# B&R Automation Studio project TD52 (part 94)

```iecst
	(* W9687 SAFETY - Room ventilation failure - Outlet air louvre group 3 - closed signal not valid *)
	xMsg9687.Enable	   		:= OUT_EG.bSafetyPLC_Active AND bRelModul_ParaSetupOk;			(* SAFETY PLC *)
	xMsg9687.Set	  		:= NOT bAMM_9687;
	xMsg9687.PT	       		:= T#0s;
	xMsg9687.Prio	   		:= 4;
	xMsg9687.RiskClass		:= 4;
	xMsg9687.Reset	   		:= FALSE;
	xMsg9687();
	MM2VIS.bMsg9687			:= xMsg9687.Q;

	(* W9688 SAFETY - Room ventilation failure - Outlet air louvre group 3 - plausibility check failure *)
	xMsg9688.Enable	   		:= OUT_EG.bSafetyPLC_Active AND bRelModul_ParaSetupOk;			(* SAFETY PLC *)
	xMsg9688.Set	  		:= NOT bAMM_9688;
	xMsg9688.PT	       		:= T#0s;
	xMsg9688.Prio	   		:= 4;
	xMsg9688.RiskClass		:= 4;
	xMsg9688.Reset	   		:= FALSE;
	xMsg9688();
	MM2VIS.bMsg9688			:= xMsg9688.Q;

	(* W9689 SAFETY - Room ventilation failure - Outlet air louvre group 4 - closed signal *)
	xMsg9689.Enable	   		:= OUT_EG.bSafetyPLC_Active AND bRelModul_ParaSetupOk;			(* SAFETY PLC *)
	xMsg9689.Set	  		:= NOT bAMM_9689;
	xMsg9689.PT	       		:= T#0s;
	xMsg9689.Prio	   		:= 4;
	xMsg9689.RiskClass		:= 4;
	xMsg9689.Reset	   		:= FALSE;
	xMsg9689();
	MM2VIS.bMsg9689			:= xMsg9689.Q;

	(* W9690 SAFETY - Room ventilation failure - Outlet air louvre group 4 - opened signal not valid *)
	xMsg9690.Enable	   		:= OUT_EG.bSafetyPLC_Active AND bRelModul_ParaSetupOk;			(* SAFETY PLC *)
	xMsg9690.Set	  		:= NOT bAMM_9690;
	xMsg9690.PT	       		:= T#0s;
	xMsg9690.Prio	   		:= 4;
	xMsg9690.RiskClass		:= 4;
	xMsg9690.Reset	   		:= FALSE;
	xMsg9690();
	MM2VIS.bMsg9690			:= xMsg9690.Q;

	(* W9691 SAFETY - Room ventilation failure - Outlet air louvre group 4 - closed signal not valid *)
	xMsg9691.Enable	   		:= OUT_EG.bSafetyPLC_Active AND bRelModul_ParaSetupOk;			(* SAFETY PLC *)
	xMsg9691.Set	  		:= NOT bAMM_9691;
	xMsg9691.PT	       		:= T#0s;
	xMsg9691.Prio	   		:= 4;
	xMsg9691.RiskClass		:= 4;
	xMsg9691.Reset	   		:= FALSE;
	xMsg9691();
	MM2VIS.bMsg9691			:= xMsg9691.Q;

	(* W9692 SAFETY - Room ventilation failure - Outlet air louvre group 4 - plausibility check failure *)
	xMsg9692.Enable	   		:= OUT_EG.bSafetyPLC_Active AND bRelModul_ParaSetupOk;			(* SAFETY PLC *)
	xMsg9692.Set	  		:= NOT bAMM_9692;
	xMsg9692.PT	       		:= T#0s;
	xMsg9692.Prio	   		:= 4;
	xMsg9692.RiskClass		:= 4;
	xMsg9692.Reset	   		:= FALSE;
	xMsg9692();
	MM2VIS.bMsg9692			:= xMsg9692.Q;

	(* W9693 SAFETY - Room ventilation failure - Outlet air louvre group 5 - closed signal *)
	xMsg9693.Enable	   		:= OUT_EG.bSafetyPLC_Active AND bRelModul_ParaSetupOk;			(* SAFETY PLC *)
	xMsg9693.Set	  		:= NOT bAMM_9693;
	xMsg9693.PT	       		:= T#0s;
	xMsg9693.Prio	   		:= 4;
	xMsg9693.RiskClass		:= 4;
	xMsg9693.Reset	   		:= FALSE;
	xMsg9693();
	MM2VIS.bMsg9693			:= xMsg9693.Q;

	(* W9694 SAFETY - Room ventilation failure - Outlet air louvre group 5 - opened signal not valid *)
	xMsg9694.Enable	   		:= OUT_EG.bSafetyPLC_Active AND bRelModul_ParaSetupOk;			(* SAFETY PLC *)
	xMsg9694.Set	  		:= NOT bAMM_9694;
	xMsg9694.PT	       		:= T#0s;
	xMsg9694.Prio	   		:= 4;
	xMsg9694.RiskClass		:= 4;
	xMsg9694.Reset	   		:= FALSE;
	xMsg9694();
	MM2VIS.bMsg9694			:= xMsg9694.Q;

	(* W9695 SAFETY - Room ventilation failure - Outlet air louvre group 5 - closed signal not valid *)
	xMsg9695.Enable	   		:= OUT_EG.bSafetyPLC_Active AND bRelModul_ParaSetupOk;			(* SAFETY PLC *)
	xMsg9695.Set	  		:= NOT bAMM_9695;
	xMsg9695.PT	       		:= T#0s;
	xMsg9695.Prio	   		:= 4;
	xMsg9695.RiskClass		:= 4;
	xMsg9695.Reset	   		:= FALSE;
	xMsg9695();
	MM2VIS.bMsg9695			:= xMsg9695.Q;

	(* W9696 SAFETY - Room ventilation failure - Outlet air louvre group 5 - plausibility check failure *)
	xMsg9696.Enable	   		:= OUT_EG.bSafetyPLC_Active AND bRelModul_ParaSetupOk;			(* SAFETY PLC *)
	xMsg9696.Set	  		:= NOT bAMM_9696;
	xMsg9696.PT	       		:= T#0s;
	xMsg9696.Prio	   		:= 4;
	xMsg9696.RiskClass		:= 4;
	xMsg9696.Reset	   		:= FALSE;
	xMsg9696();
	MM2VIS.bMsg9696			:= xMsg9696.Q;

	(* W9697 SAFETY - Room ventilation failure - Outlet air louvre group 6 - closed signal *)
	xMsg9697.Enable	   		:= OUT_EG.bSafetyPLC_Active AND bRelModul_ParaSetupOk;			(* SAFETY PLC *)
	xMsg9697.Set	  		:= NOT bAMM_9697;
	xMsg9697.PT	       		:= T#0s;
	xMsg9697.Prio	   		:= 4;
	xMsg9697.RiskClass		:= 4;
	xMsg9697.Reset	   		:= FALSE;
	xMsg9697();
	MM2VIS.bMsg9697			:= xMsg9697.Q;

	(* W9698 SAFETY - Room ventilation failure - Outlet air louvre group 6 - opened signal not valid *)
	xMsg9698.Enable	   		:= OUT_EG.bSafetyPLC_Active AND bRelModul_ParaSetupOk;			(* SAFETY PLC *)
	xMsg9698.Set	  		:= NOT bAMM_9698;
	xMsg9698.PT	       		:= T#0s;
	xMsg9698.Prio	   		:= 4;
	xMsg9698.RiskClass		:= 4;
	xMsg9698.Reset	   		:= FALSE;
	xMsg9698();
	MM2VIS.bMsg9698			:= xMsg9698.Q;

	(* W9699 SAFETY - Room ventilation failure - Outlet air louvre group 6 - closed signal not valid *)
	xMsg9699.Enable	   		:= OUT_EG.bSafetyPLC_Active AND bRelModul_ParaSetupOk;			(* SAFETY PLC *)
	xMsg9699.Set	  		:= NOT bAMM_9699;
	xMsg9699.PT	       		:= T#0s;
	xMsg9699.Prio	   		:= 4;
	xMsg9699.RiskClass		:= 4;
	xMsg9699.Reset	   		:= FALSE;
	xMsg9699();
	MM2VIS.bMsg9699			:= xMsg9699.Q;

	(* W9700 SAFETY - Room ventilation failure - Outlet air louvre group 6 - plausibility check failure *)
	xMsg9700.Enable	   		:= OUT_EG.bSafetyPLC_Active AND bRelModul_ParaSetupOk;			(* SAFETY PLC *)
	xMsg9700.Set	  		:= NOT bAMM_9700;
	xMsg9700.PT	       		:= T#0s;
	xMsg9700.Prio	   		:= 4;
	xMsg9700.RiskClass		:= 4;
	xMsg9700.Reset	   		:= FALSE;
	xMsg9700();
	MM2VIS.bMsg9700			:= xMsg9700.Q;

	(* W9701 SAFETY - Release gas valve A for decentral gas addition - output not valid *)
	xMsg9701.Enable	   		:= OUT_EG.bSafetyPLC_Active AND bRelModul_ParaSetupOk;			(* SAFETY PLC *)
	xMsg9701.Set	  		:= NOT bAMM_9701;
	xMsg9701.PT	       		:= T#0s;
	xMsg9701.Prio	   		:= 4;
	xMsg9701.RiskClass		:= 4;
	xMsg9701.Reset	   		:= FALSE;
	xMsg9701();
	MM2VIS.bMsg9701			:= xMsg9701.Q;

	(* W9702 SAFETY - Release gas valve B for decentral gas addition - output not valid *)
	xMsg9702.Enable	   		:= OUT_EG.bSafetyPLC_Active AND bRelModul_ParaSetupOk;			(* SAFETY PLC *)
	xMsg9702.Set	  		:= NOT bAMM_9702;
	xMsg9702.PT	       		:= T#0s;
	xMsg9702.Prio	   		:= 4;
	xMsg9702.RiskClass		:= 4;
	xMsg9702.Reset	   		:= FALSE;
	xMsg9702();
	MM2VIS.bMsg9702			:= xMsg9702.Q;

	(* W9703 SAFETY - Gas safety device for decentral gas addition - signal not valid *)
	xMsg9703.Enable	   		:= OUT_EG.bSafetyPLC_Active AND bRelModul_ParaSetupOk;			(* SAFETY PLC *)
	xMsg9703.Set	  		:= NOT bAMM_9703;
	xMsg9703.PT	       		:= T#0s;
	xMsg9703.Prio	   		:= 4;
	xMsg9703.RiskClass		:= 4;
	xMsg9703.Reset	   		:= FALSE;
	xMsg9703();
	MM2VIS.bMsg9703			:= xMsg9703.Q;

	(* W9704 SAFETY - Gas safety device for decentral gas addition - output not valid *)
	xMsg9704.Enable	   		:= OUT_EG.bSafetyPLC_Active AND bRelModul_ParaSetupOk;			(* SAFETY PLC *)
	xMsg9704.Set	  		:= NOT bAMM_9704;
	xMsg9704.PT	       		:= T#0s;
	xMsg9704.Prio	   		:= 4;
	xMsg9704.RiskClass		:= 4;
	xMsg9704.Reset	   		:= FALSE;
	xMsg9704();
	MM2VIS.bMsg9704			:= xMsg9704.Q;

	(*---------------------------------------------------------------------------*)
	(* operating messages > AMM *)

	(* B2190 Emergency stop push button - module control panel (+A/+MC) *)
	xMsg2190.Enable		:= NOT OUT_EG.bSafetyPLC_Active AND bRelModul_ParaSetupOk;			(* SAFETY PLC *)
	xMsg2190.Set		:= IN_EG.tEmStop_MC.Di;
	xMsg2190.Reset		:= TRUE;
	xMsg2190();
	MM2VIS.bMsg2190		:= xMsg2190.Q;

	(* B2191 Emergency stop push button - module interface panel (+M) *)
	xMsg2191.Enable		:= NOT OUT_EG.bSafetyPLC_Active AND bRelModul_ParaSetupOk;			(* SAFETY PLC *)
	xMsg2191.Set		:= IN_EG.tEmStop_M.Di;
	xMsg2191.Reset		:= TRUE;
	xMsg2191();
	MM2VIS.bMsg2191		:= xMsg2191.Q;

	(* B2192 Emergency stop push button – master control panel (+ST) *)
	xMsg2192.Enable		:= NOT OUT_EG.bSafetyPLC_Active AND bRelModul_ParaSetupOk;			(* SAFETY PLC *)
	xMsg2192.Set		:= IN_EG.tEmStop_ST.Di;
	xMsg2192.Reset		:= TRUE;
	xMsg2192();
	MM2VIS.bMsg2192		:= xMsg2192.Q;

	(* B2193 Emergency stop push button – interlock panel (+IS) *)
	xMsg2193.Enable		:= NOT OUT_EG.bSafetyPLC_Active AND bRelModul_ParaSetupOk;			(* SAFETY PLC *)
	xMsg2193.Set		:= IN_EG.tEmStop_IS.Di;
	xMsg2193.Reset		:= TRUE;
	xMsg2193();
	MM2VIS.bMsg2193		:= xMsg2193.Q;

	(* B2194 Emergency stop push button – thermal reactor control panel (+TS) *)
	xMsg2194.Enable		:= NOT OUT_EG.bSafetyPLC_Active AND bRelModul_ParaSetupOk;			(* SAFETY PLC *)
	xMsg2194.Set		:= IN_EG.tEmStop_TS.Di;
	xMsg2194.Reset		:= TRUE;
	xMsg2194();
	MM2VIS.bMsg2194		:= xMsg2194.Q;

	(* B2195 Emergency stop push button – generator interface panel (+GENI) *)
	xMsg2195.Enable		:= NOT OUT_EG.bSafetyPLC_Active AND bRelModul_ParaSetupOk;			(* SAFETY PLC *)
	xMsg2195.Set		:= IN_EG.tEmStop_GENI.Di;
	xMsg2195.Reset		:= TRUE;
	xMsg2195();
	MM2VIS.bMsg2195		:= xMsg2195.Q;

	(* B2196 Emergency stop push button – engine interface panel bank A (+ENGIA) *)
	xMsg2196.Enable		:= NOT OUT_EG.bSafetyPLC_Active AND bRelModul_ParaSetupOk;			(* SAFETY PLC *)
	xMsg2196.Set		:= IN_EG.tEmStop_ENGIA.Di;
	xMsg2196.Reset		:= TRUE;
	xMsg2196();
	MM2VIS.bMsg2196		:= xMsg2196.Q;

	(* B2197 Emergency stop push button – turbocharger module interface panel (+TCMI) *)
	xMsg2197.Enable		:= NOT OUT_EG.bSafetyPLC_Active AND bRelModul_ParaSetupOk;			(* SAFETY PLC *)
	xMsg2197.Set		:= IN_EG.tEmStop_TCMI.Di;
	xMsg2197.Reset		:= TRUE;
	xMsg2197();
	MM2VIS.bMsg2197		:= xMsg2197.Q;

	(* B2198 Emergency stop push button – jacket water module interface panel (+JWMI) *)
	xMsg2198.Enable		:= NOT OUT_EG.bSafetyPLC_Active AND bRelModul_ParaSetupOk;			(* SAFETY PLC *)
	xMsg2198.Set		:= IN_EG.tEmStop_JWMI.Di;
	xMsg2198.Reset		:= TRUE;
	xMsg2198();
	MM2VIS.bMsg2198		:= xMsg2198.Q;

	(* B2199 Emergency stop push button – oil module interface panel (+OILMI) *)
	xMsg2199.Enable		:= NOT OUT_EG.bSafetyPLC_Active AND bRelModul_ParaSetupOk;			(* SAFETY PLC *)
	xMsg2199.Set		:= IN_EG.tEmStop_OILMI.Di;
	xMsg2199.Reset		:= TRUE;
	xMsg2199();
	MM2VIS.bMsg2199		:= xMsg2199.Q;

	(* B2200 Emergency stop push button – exhaust gas after treatment control panel (+SCR) *)
	xMsg2200.Enable		:= NOT OUT_EG.bSafetyPLC_Active AND bRelModul_ParaSetupOk;			(* SAFETY PLC *)
	xMsg2200.Set		:= IN_EG.tEmStop_SCR.Di;
	xMsg2200.Reset		:= TRUE;
	xMsg2200();
	MM2VIS.bMsg2200		:= xMsg2200.Q;

	(* B2804 measuring signal failure main bearing temperature xx *)
	xMsg2804.Enable		:= TRUE;
	xMsg2804.Set		:= bOpM_T_MBearing_Ms;
	xMsg2804.Reset		:= TRUE;
	xMsg2804();
	MM2VIS.bMsg2804		:= xMsg2804.Q;

	(* B2805 main bearing temperature high *)
	xMsg2805.Enable		:= TRUE;
	xMsg2805.Set		:= bOpM_T_MBearing_Hi;
	xMsg2805.Reset		:= TRUE;
	xMsg2805();
	MM2VIS.bMsg2805		:= xMsg2805.Q;

	(* B2806 measuring signal failure conrod bearing temperature xx *)
	xMsg2806.Enable		:= TRUE;
	xMsg2806.Set		:= bOpM_T_CBearing_Ms;
	xMsg2806.Reset		:= TRUE;
	xMsg2806();
	MM2VIS.bMsg2806		:= xMsg2806.Q;

	(* B2807 conrod bearing temperature high *)
	xMsg2807.Enable		:= TRUE;
	xMsg2807.Set		:= bOpM_T_CBearing_Hi;
	xMsg2807.Reset		:= TRUE;
	xMsg2807();
	MM2VIS.bMsg2807		:= xMsg2807.Q;

	(* B2822 conrod bearing signal intensity minimum *)
	xMsg2822.Enable		:= TRUE;
	xMsg2822.Set		:= bOpM_T_CBearing_Sig_Lo;
	xMsg2822.Reset		:= TRUE;
	xMsg2822();
	MM2VIS.bMsg2822		:= xMsg2822.Q;

	(* B2904 main bearing temperature - positive MEDIAN deviation maximum *)
	xMsg2904.Enable		:= TRUE;
	xMsg2904.Set		:= bOpM_T_MBearing_MDev_HiHi;
	xMsg2904.Reset		:= TRUE;
	xMsg2904();
	MM2VIS.bMsg2904		:= xMsg2904.Q;

	(* B2905 conrod bearing temperature - positive MEDIAN deviation maximum *)
	xMsg2905.Enable		:= TRUE;
	xMsg2905.Set		:= bOpM_T_CBearing_MDev_HiHi;
	xMsg2905.Reset		:= TRUE;
	xMsg2905();
	MM2VIS.bMsg2905		:= xMsg2905.Q;

	(* B2909 Conrod bearing temperature calibration successful *)
	xTOF_Calib_Ok(IN 	:= bOpM_T_CBearing_Calib_Ok, PT := T#1s);		(* increase message time from 100ms to 1 s for HMI *)

	xMsg2909.Enable		:= TRUE;
	xMsg2909.Set		:= xTOF_Calib_Ok.Q;
	xMsg2909.Reset		:= TRUE;
	xMsg2909();
	MM2VIS.bMsg2909		:= xMsg2909.Q;

	(* B2958 main bearing temperature - negative MEDIAN deviation maximum *)
	xMsg2958.Enable		:= TRUE;
	xMsg2958.Set		:= bOpM_T_MBearing_MDev_Lo;
	xMsg2958.Reset		:= TRUE;
	xMsg2958();
	MM2VIS.bMsg2958		:= xMsg2958.Q;

	(* B2959 conrod bearing temperature - negative MEDIAN deviation maximum *)
	xMsg2959.Enable		:= TRUE;
	xMsg2959.Set		:= bOpM_T_CBearing_MDev_Lo;
	xMsg2959.Reset		:= TRUE;
	xMsg2959();
	MM2VIS.bMsg2959		:= xMsg2959.Q;

	(* B2981 PU scuffing detection *)
	xMsg2981.Enable		:= Para.bPUscf_Ena;
	xMsg2981.Set		:= bOpM_PUscuff AND bAMM_PUscuff;
	xMsg2981.Reset		:= TRUE;
	xMsg2981();
	MM2VIS.bMsg2981		:= xMsg2981.Q;

	(* B9038 Emergency stop push button – exhaust gas scavenging system control panel (+TCMSCAV) *)
	xMsg9038.Enable		:= NOT OUT_EG.bSafetyPLC_Active AND bRelModul_ParaSetupOk;			(* SAFETY PLC *)
	xMsg9038.Set		:= IN_EG.tEmStop_TCMSCAV.Di;
	xMsg9038.Reset		:= TRUE;
	xMsg9038();
	MM2VIS.bMsg9038		:= xMsg9038.Q;

	(*---------------------------------------------------------------------------*)
	(* general alarms for further module operations *)
	bGnlTrip1 	:= OUT_EG.tEG2AB.bGnlTrip1 		OR IN_EG.tAB2EG.bGnlTrip1;
	bGnlTrip2 	:= OUT_EG.tEG2AB.bGnlTrip2 		OR IN_EG.tAB2EG.bGnlTrip2;
	bGnlTrip3 	:= OUT_EG.tEG2AB.bGnlTrip3 		OR IN_EG.tAB2EG.bGnlTrip3;
	bGnlWarning := OUT_EG.tEG2AB.bGnlWarning	OR IN_EG.tAB2EG.bGnlWarning;
	bGnlTrip	:= bGnlTrip1 OR bGnlTrip2 OR bGnlTrip3;
	(*****************************************************************************)
END_PROGRAM
```

#### MsgEGInit.st - Cyclic code
```iecst
(*******************************************************************************
Msg_EG	 			 alarms generation MM_EngineGeneral

This code is confidential and proprietary to the INNIO Company.
It may not be used in any form, or reproduced in any manner,
without written permission of the INNIO Company.
Copyright, INNIO Company, 2019

Instructions FOR use:
--------------------
1) declare alarm with function block "Msg"

2) use template to create a new alarm, substitue 0000 by message number:

	xMsg0000.Num		:=	0000;					alarm number
	xMsg0000.AmmSysAdr	:=  iAdrAmmBase2MM;			do not change
	xMsg0000.AmmOutAdr	:=  iAdrMM2AmmBase;			do not change

3) 	set alarm number

(*******************************************************************************)
PROGRAM _INIT

	iAdrAmmBase2MM		:= ADR(IN_EG.tAB2EG);
	iAdrMM2AmmBase		:= ADR(OUT_EG.tEG2AB);

	(*---------------------------------------------------------------------------*)

	xMsg1026.Num		:= 1026;
	xMsg1026.AmmInAdr	:= iAdrAmmBase2MM;
	xMsg1026.AmmOutAdr	:= iAdrMM2AmmBase;

	xMsg1031.Num		:= 1031;
	xMsg1031.AmmInAdr	:= iAdrAmmBase2MM;
	xMsg1031.AmmOutAdr	:= iAdrMM2AmmBase;

	xMsg1056.Num		:= 1056;
	xMsg1056.AmmInAdr	:= iAdrAmmBase2MM;
	xMsg1056.AmmOutAdr	:= iAdrMM2AmmBase;

	xMsg1168.Num		:= 1168;
	xMsg1168.AmmInAdr	:= iAdrAmmBase2MM;
	xMsg1168.AmmOutAdr	:= iAdrMM2AmmBase;

	xMsg2190.Num		:= 2190;
	xMsg2190.AmmInAdr	:= iAdrAmmBase2MM;
	xMsg2190.AmmOutAdr	:= iAdrMM2AmmBase;

	xMsg2191.Num		:= 2191;
	xMsg2191.AmmInAdr	:= iAdrAmmBase2MM;
	xMsg2191.AmmOutAdr	:= iAdrMM2AmmBase;

	xMsg2192.Num		:= 2192;
	xMsg2192.AmmInAdr	:= iAdrAmmBase2MM;
	xMsg2192.AmmOutAdr	:= iAdrMM2AmmBase;

	xMsg2193.Num		:= 2193;
	xMsg2193.AmmInAdr	:= iAdrAmmBase2MM;
	xMsg2193.AmmOutAdr	:= iAdrMM2AmmBase;

	xMsg2194.Num		:= 2194;
	xMsg2194.AmmInAdr	:= iAdrAmmBase2MM;
	xMsg2194.AmmOutAdr	:= iAdrMM2AmmBase;

	xMsg2195.Num		:= 2195;
	xMsg2195.AmmInAdr	:= iAdrAmmBase2MM;
	xMsg2195.AmmOutAdr	:= iAdrMM2AmmBase;

	xMsg2196.Num		:= 2196;
	xMsg2196.AmmInAdr	:= iAdrAmmBase2MM;
	xMsg2196.AmmOutAdr	:= iAdrMM2AmmBase;

	xMsg2197.Num		:= 2197;
	xMsg2197.AmmInAdr	:= iAdrAmmBase2MM;
	xMsg2197.AmmOutAdr	:= iAdrMM2AmmBase;

	xMsg2198.Num		:= 2198;
	xMsg2198.AmmInAdr	:= iAdrAmmBase2MM;
	xMsg2198.AmmOutAdr	:= iAdrMM2AmmBase;

	xMsg2199.Num		:= 2199;
	xMsg2199.AmmInAdr	:= iAdrAmmBase2MM;
	xMsg2199.AmmOutAdr	:= iAdrMM2AmmBase;

	xMsg2200.Num		:= 2200;
	xMsg2200.AmmInAdr	:= iAdrAmmBase2MM;
	xMsg2200.AmmOutAdr	:= iAdrMM2AmmBase;

	xMsg2227.Num		:= 2227;
	xMsg2227.AmmInAdr	:= iAdrAmmBase2MM;
	xMsg2227.AmmOutAdr	:= iAdrMM2AmmBase;

	xMsg2228.Num		:= 2228;
	xMsg2228.AmmInAdr	:= iAdrAmmBase2MM;
	xMsg2228.AmmOutAdr	:= iAdrMM2AmmBase;

	xMsg2229.Num		:= 2229;
	xMsg2229.AmmInAdr	:= iAdrAmmBase2MM;
	xMsg2229.AmmOutAdr	:= iAdrMM2AmmBase;

	xMsg2230.Num		:= 2230;
	xMsg2230.AmmInAdr	:= iAdrAmmBase2MM;
	xMsg2230.AmmOutAdr	:= iAdrMM2AmmBase;

	xMsg2232.Num		:= 2232;
	xMsg2232.AmmInAdr	:= iAdrAmmBase2MM;
	xMsg2232.AmmOutAdr	:= iAdrMM2AmmBase;

	xMsg2270.Num		:= 2270;
	xMsg2270.AmmInAdr	:= iAdrAmmBase2MM;
	xMsg2270.AmmOutAdr	:= iAdrMM2AmmBase;

	xMsg2285.Num		:= 2285;
	xMsg2285.AmmInAdr	:= iAdrAmmBase2MM;
	xMsg2285.AmmOutAdr	:= iAdrMM2AmmBase;

	xMsg2286.Num		:= 2286;
	xMsg2286.AmmInAdr	:= iAdrAmmBase2MM;
	xMsg2286.AmmOutAdr	:= iAdrMM2AmmBase;

	xMsg2300.Num		:= 2300;
	xMsg2300.AmmInAdr	:= iAdrAmmBase2MM;
	xMsg2300.AmmOutAdr	:= iAdrMM2AmmBase;

	xMsg2362.Num		:= 2362;
	xMsg2362.AmmInAdr	:= iAdrAmmBase2MM;
	xMsg2362.AmmOutAdr	:= iAdrMM2AmmBase;

	xMsg2383.Num		:= 2383;
	xMsg2383.AmmInAdr	:= iAdrAmmBase2MM;
	xMsg2383.AmmOutAdr	:= iAdrMM2AmmBase;

	xMsg2384.Num		:= 2384;
	xMsg2384.AmmInAdr	:= iAdrAmmBase2MM;
	xMsg2384.AmmOutAdr	:= iAdrMM2AmmBase;

	xMsg2385.Num		:= 2385;
	xMsg2385.AmmInAdr	:= iAdrAmmBase2MM;
	xMsg2385.AmmOutAdr	:= iAdrMM2AmmBase;

	xMsg2386.Num		:= 2386;
	xMsg2386.AmmInAdr	:= iAdrAmmBase2MM;
	xMsg2386.AmmOutAdr	:= iAdrMM2AmmBase;

	xMsg2387.Num		:= 2387;
	xMsg2387.AmmInAdr	:= iAdrAmmBase2MM;
	xMsg2387.AmmOutAdr	:= iAdrMM2AmmBase;

	xMsg2388.Num		:= 2388;
	xMsg2388.AmmInAdr	:= iAdrAmmBase2MM;
	xMsg2388.AmmOutAdr	:= iAdrMM2AmmBase;

	xMsg2389.Num		:= 2389;
	xMsg2389.AmmInAdr	:= iAdrAmmBase2MM;
	xMsg2389.AmmOutAdr	:= iAdrMM2AmmBase;

	xMsg2390.Num		:= 2390;
	xMsg2390.AmmInAdr	:= iAdrAmmBase2MM;
	xMsg2390.AmmOutAdr	:= iAdrMM2AmmBase;

	xMsg2391.Num		:= 2391;
	xMsg2391.AmmInAdr	:= iAdrAmmBase2MM;
	xMsg2391.AmmOutAdr	:= iAdrMM2AmmBase;

	xMsg2392.Num		:= 2392;
	xMsg2392.AmmInAdr	:= iAdrAmmBase2MM;
	xMsg2392.AmmOutAdr	:= iAdrMM2AmmBase;

	xMsg2393.Num		:= 2393;
	xMsg2393.AmmInAdr	:= iAdrAmmBase2MM;
	xMsg2393.AmmOutAdr	:= iAdrMM2AmmBase;

	xMsg2394.Num		:= 2394;
	xMsg2394.AmmInAdr	:= iAdrAmmBase2MM;
	xMsg2394.AmmOutAdr	:= iAdrMM2AmmBase;

	xMsg2395.Num		:= 2395;
	xMsg2395.AmmInAdr	:= iAdrAmmBase2MM;
	xMsg2395.AmmOutAdr	:= iAdrMM2AmmBase;

	xMsg2396.Num		:= 2396;
	xMsg2396.AmmInAdr	:= iAdrAmmBase2MM;
	xMsg2396.AmmOutAdr	:= iAdrMM2AmmBase;

	xMsg2397.Num		:= 2397;
	xMsg2397.AmmInAdr	:= iAdrAmmBase2MM;
	xMsg2397.AmmOutAdr	:= iAdrMM2AmmBase;

	xMsg2398.Num		:= 2398;
	xMsg2398.AmmInAdr	:= iAdrAmmBase2MM;
	xMsg2398.AmmOutAdr	:= iAdrMM2AmmBase;

	xMsg2542.Num		:= 2542;
	xMsg2542.AmmInAdr	:= iAdrAmmBase2MM;
	xMsg2542.AmmOutAdr	:= iAdrMM2AmmBase;

	xMsg2544.Num		:= 2544;
	xMsg2544.AmmInAdr	:= iAdrAmmBase2MM;
	xMsg2544.AmmOutAdr	:= iAdrMM2AmmBase;

	xMsg2552.Num		:= 2552;
	xMsg2552.AmmInAdr	:= iAdrAmmBase2MM;
	xMsg2552.AmmOutAdr	:= iAdrMM2AmmBase;

	xMsg2553.Num		:= 2553;
	xMsg2553.AmmInAdr	:= iAdrAmmBase2MM;
	xMsg2553.AmmOutAdr	:= iAdrMM2AmmBase;

	xMsg2561.Num		:= 2561;
	xMsg2561.AmmInAdr	:= iAdrAmmBase2MM;
	xMsg2561.AmmOutAdr	:= iAdrMM2AmmBase;

	xMsg2790.Num		:= 2790;
	xMsg2790.AmmInAdr	:= iAdrAmmBase2MM;
	xMsg2790.AmmOutAdr	:= iAdrMM2AmmBase;

	xMsg2794.Num		:= 2794;
	xMsg2794.AmmInAdr	:= iAdrAmmBase2MM;
	xMsg2794.AmmOutAdr	:= iAdrMM2AmmBase;

	xMsg2804.Num		:= 2804;
	xMsg2804.AmmInAdr	:= iAdrAmmBase2MM;
	xMsg2804.AmmOutAdr	:= iAdrMM2AmmBase;

	xMsg2805.Num		:= 2805;
	xMsg2805.AmmInAdr	:= iAdrAmmBase2MM;
	xMsg2805.AmmOutAdr	:= iAdrMM2AmmBase;

	xMsg2806.Num		:= 2806;
	xMsg2806.AmmInAdr	:= iAdrAmmBase2MM;
	xMsg2806.AmmOutAdr	:= iAdrMM2AmmBase;

	xMsg2807.Num		:= 2807;
	xMsg2807.AmmInAdr	:= iAdrAmmBase2MM;
	xMsg2807.AmmOutAdr	:= iAdrMM2AmmBase;

	xMsg2822.Num		:= 2822;
	xMsg2822.AmmInAdr	:= iAdrAmmBase2MM;
	xMsg2822.AmmOutAdr	:= iAdrMM2AmmBase;

	xMsg2904.Num		:= 2904;
	xMsg2904.AmmInAdr	:= iAdrAmmBase2MM;
	xMsg2904.AmmOutAdr	:= iAdrMM2AmmBase;

	xMsg2905.Num		:= 2905;
	xMsg2905.AmmInAdr	:= iAdrAmmBase2MM;
	xMsg2905.AmmOutAdr	:= iAdrMM2AmmBase;

	xMsg2909.Num		:= 2909;
	xMsg2909.AmmInAdr	:= iAdrAmmBase2MM;
	xMsg2909.AmmOutAdr	:= iAdrMM2AmmBase;

	xMsg2958.Num		:= 2958;
	xMsg2958.AmmInAdr	:= iAdrAmmBase2MM;
	xMsg2958.AmmOutAdr	:= iAdrMM2AmmBase;

	xMsg2959.Num		:= 2959;
	xMsg2959.AmmInAdr	:= iAdrAmmBase2MM;
	xMsg2959.AmmOutAdr	:= iAdrMM2AmmBase;

	xMsg2981.Num		:= 2981;
	xMsg2981.AmmInAdr	:= iAdrAmmBase2MM;
	xMsg2981.AmmOutAdr	:= iAdrMM2AmmBase;

	xMsg3368.Num		:= 3368;
	xMsg3368.AmmInAdr	:= iAdrAmmBase2MM;
	xMsg3368.AmmOutAdr	:= iAdrMM2AmmBase;

	xMsg3378.Num		:= 3378;
	xMsg3378.AmmInAdr	:= iAdrAmmBase2MM;
	xMsg3378.AmmOutAdr	:= iAdrMM2AmmBase;

	xMsg3396.Num		:= 3396;
	xMsg3396.AmmInAdr	:= iAdrAmmBase2MM;
	xMsg3396.AmmOutAdr	:= iAdrMM2AmmBase;

	xMsg3449.Num		:= 3449;
	xMsg3449.AmmInAdr	:= iAdrAmmBase2MM;
	xMsg3449.AmmOutAdr	:= iAdrMM2AmmBase;

	xMsg3559.Num		:= 3559;
	xMsg3559.AmmInAdr	:= iAdrAmmBase2MM;
	xMsg3559.AmmOutAdr	:= iAdrMM2AmmBase;

	xMsg9038.Num		:= 9038;
	xMsg9038.AmmInAdr	:= iAdrAmmBase2MM;
	xMsg9038.AmmOutAdr	:= iAdrMM2AmmBase;

	xMsg9217.Num		:= 9217;
	xMsg9217.AmmInAdr	:= iAdrAmmBase2MM;
	xMsg9217.AmmOutAdr	:= iAdrMM2AmmBase;

	xMsg9218.Num		:= 9218;
	xMsg9218.AmmInAdr	:= iAdrAmmBase2MM;
	xMsg9218.AmmOutAdr	:= iAdrMM2AmmBase;

	xMsg9219.Num		:= 9219;
	xMsg9219.AmmInAdr	:= iAdrAmmBase2MM;
	xMsg9219.AmmOutAdr	:= iAdrMM2AmmBase;

	xMsg9408.Num		:= 9408;
	xMsg9408.AmmInAdr	:= iAdrAmmBase2MM;
	xMsg9408.AmmOutAdr	:= iAdrMM2AmmBase;

	xMsg9409.Num		:= 9409;
	xMsg9409.AmmInAdr	:= iAdrAmmBase2MM;
	xMsg9409.AmmOutAdr	:= iAdrMM2AmmBase;

	xMsg9410.Num		:= 9410;
	xMsg9410.AmmInAdr	:= iAdrAmmBase2MM;
	xMsg9410.AmmOutAdr	:= iAdrMM2AmmBase;

	xMsg9411.Num		:= 9411;
	xMsg9411.AmmInAdr	:= iAdrAmmBase2MM;
	xMsg9411.AmmOutAdr	:= iAdrMM2AmmBase;

	xMsg9412.Num		:= 9412;
	xMsg9412.AmmInAdr	:= iAdrAmmBase2MM;
	xMsg9412.AmmOutAdr	:= iAdrMM2AmmBase;

	xMsg9413.Num		:= 9413;
	xMsg9413.AmmInAdr	:= iAdrAmmBase2MM;
	xMsg9413.AmmOutAdr	:= iAdrMM2AmmBase;

	xMsg9414.Num		:= 9414;
	xMsg9414.AmmInAdr	:= iAdrAmmBase2MM;
	xMsg9414.AmmOutAdr	:= iAdrMM2AmmBase;

	xMsg9415.Num		:= 9415;
	xMsg9415.AmmInAdr	:= iAdrAmmBase2MM;
	xMsg9415.AmmOutAdr	:= iAdrMM2AmmBase;

	xMsg9416.Num		:= 9416;
	xMsg9416.AmmInAdr	:= iAdrAmmBase2MM;
	xMsg9416.AmmOutAdr	:= iAdrMM2AmmBase;

	xMsg9417.Num		:= 9417;
	xMsg9417.AmmInAdr	:= iAdrAmmBase2MM;
	xMsg9417.AmmOutAdr	:= iAdrMM2AmmBase;

	xMsg9418.Num		:= 9418;
	xMsg9418.AmmInAdr	:= iAdrAmmBase2MM;
	xMsg9418.AmmOutAdr	:= iAdrMM2AmmBase;

	xMsg9419.Num		:= 9419;
	xMsg9419.AmmInAdr	:= iAdrAmmBase2MM;
	xMsg9419.AmmOutAdr	:= iAdrMM2AmmBase;

	xMsg9420.Num		:= 9420;
	xMsg9420.AmmInAdr	:= iAdrAmmBase2MM;
	xMsg9420.AmmOutAdr	:= iAdrMM2AmmBase;

	xMsg9421.Num		:= 9421;
	xMsg9421.AmmInAdr	:= iAdrAmmBase2MM;
	xMsg9421.AmmOutAdr	:= iAdrMM2AmmBase;

	xMsg9422.Num		:= 9422;
	xMsg9422.AmmInAdr	:= iAdrAmmBase2MM;
	xMsg9422.AmmOutAdr	:= iAdrMM2AmmBase;

	xMsg9423.Num		:= 9423;
	xMsg9423.AmmInAdr	:= iAdrAmmBase2MM;
	xMsg9423.AmmOutAdr	:= iAdrMM2AmmBase;

	xMsg9424.Num		:= 9424;
	xMsg9424.AmmInAdr	:= iAdrAmmBase2MM;
	xMsg9424.AmmOutAdr	:= iAdrMM2AmmBase;

	xMsg9425.Num		:= 9425;
	xMsg9425.AmmInAdr	:= iAdrAmmBase2MM;
	xMsg9425.AmmOutAdr	:= iAdrMM2AmmBase;

	xMsg9426.Num		:= 9426;
	xMsg9426.AmmInAdr	:= iAdrAmmBase2MM;
	xMsg9426.AmmOutAdr	:= iAdrMM2AmmBase;

	xMsg9427.Num		:= 9427;
	xMsg9427.AmmInAdr	:= iAdrAmmBase2MM;
	xMsg9427.AmmOutAdr	:= iAdrMM2AmmBase;

	xMsg9428.Num		:= 9428;
	xMsg9428.AmmInAdr	:= iAdrAmmBase2MM;
	xMsg9428.AmmOutAdr	:= iAdrMM2AmmBase;

	xMsg9429.Num		:= 9429;
	xMsg9429.AmmInAdr	:= iAdrAmmBase2MM;
	xMsg9429.AmmOutAdr	:= iAdrMM2AmmBase;

	xMsg9430.Num		:= 9430;
	xMsg9430.AmmInAdr	:= iAdrAmmBase2MM;
	xMsg9430.AmmOutAdr	:= iAdrMM2AmmBase;

	xMsg9431.Num		:= 9431;
	xMsg9431.AmmInAdr	:= iAdrAmmBase2MM;
	xMsg9431.AmmOutAdr	:= iAdrMM2AmmBase;

	xMsg9433.Num		:= 9433;
	xMsg9433.AmmInAdr	:= iAdrAmmBase2MM;
	xMsg9433.AmmOutAdr	:= iAdrMM2AmmBase;

	xMsg9434.Num		:= 9434;
	xMsg9434.AmmInAdr	:= iAdrAmmBase2MM;
	xMsg9434.AmmOutAdr	:= iAdrMM2AmmBase;

	xMsg9437.Num		:= 9437;
	xMsg9437.AmmInAdr	:= iAdrAmmBase2MM;
	xMsg9437.AmmOutAdr	:= iAdrMM2AmmBase;

	xMsg9438.Num		:= 9438;
	xMsg9438.AmmInAdr	:= iAdrAmmBase2MM;
	xMsg9438.AmmOutAdr	:= iAdrMM2AmmBase;

	xMsg9439.Num		:= 9439;
	xMsg9439.AmmInAdr	:= iAdrAmmBase2MM;
	xMsg9439.AmmOutAdr	:= iAdrMM2AmmBase;

	xMsg9440.Num		:= 9440;
	xMsg9440.AmmInAdr	:= iAdrAmmBase2MM;
	xMsg9440.AmmOutAdr	:= iAdrMM2AmmBase;

	xMsg9441.Num		:= 9441;
	xMsg9441.AmmInAdr	:= iAdrAmmBase2MM;
	xMsg9441.AmmOutAdr	:= iAdrMM2AmmBase;

	xMsg9442.Num		:= 9442;
	xMsg9442.AmmInAdr	:= iAdrAmmBase2MM;
	xMsg9442.AmmOutAdr	:= iAdrMM2AmmBase;

	xMsg9443.Num		:= 9443;
	xMsg9443.AmmInAdr	:= iAdrAmmBase2MM;
	xMsg9443.AmmOutAdr	:= iAdrMM2AmmBase;

	xMsg9444.Num		:= 9444;
	xMsg9444.AmmInAdr	:= iAdrAmmBase2MM;
	xMsg9444.AmmOutAdr	:= iAdrMM2AmmBase;

	xMsg9445.Num		:= 9445;
	xMsg9445.AmmInAdr	:= iAdrAmmBase2MM;
	xMsg9445.AmmOutAdr	:= iAdrMM2AmmBase;

	xMsg9446.Num		:= 9446;
	xMsg9446.AmmInAdr	:= iAdrAmmBase2MM;
	xMsg9446.AmmOutAdr	:= iAdrMM2AmmBase;

	xMsg9447.Num		:= 9447;
	xMsg9447.AmmInAdr	:= iAdrAmmBase2MM;
	xMsg9447.AmmOutAdr	:= iAdrMM2AmmBase;

	xMsg9448.Num		:= 9448;
	xMsg9448.AmmInAdr	:= iAdrAmmBase2MM;
	xMsg9448.AmmOutAdr	:= iAdrMM2AmmBase;

	xMsg9449.Num		:= 9449;
	xMsg9449.AmmInAdr	:= iAdrAmmBase2MM;
	xMsg9449.AmmOutAdr	:= iAdrMM2AmmBase;

	xMsg9450.Num		:= 9450;
	xMsg9450.AmmInAdr	:= iAdrAmmBase2MM;
	xMsg9450.AmmOutAdr	:= iAdrMM2AmmBase;

	xMsg9451.Num		:= 9451;
	xMsg9451.AmmInAdr	:= iAdrAmmBase2MM;
	xMsg9451.AmmOutAdr	:= iAdrMM2AmmBase;

	xMsg9452.Num		:= 9452;
	xMsg9452.AmmInAdr	:= iAdrAmmBase2MM;
	xMsg9452.AmmOutAdr	:= iAdrMM2AmmBase;

	xMsg9453.Num		:= 9453;
	xMsg9453.AmmInAdr	:= iAdrAmmBase2MM;
	xMsg9453.AmmOutAdr	:= iAdrMM2AmmBase;

	xMsg9454.Num		:= 9454;
	xMsg9454.AmmInAdr	:= iAdrAmmBase2MM;
	xMsg9454.AmmOutAdr	:= iAdrMM2AmmBase;

	xMsg9455.Num		:= 9455;
	xMsg9455.AmmInAdr	:= iAdrAmmBase2MM;
	xMsg9455.AmmOutAdr	:= iAdrMM2AmmBase;

	xMsg9456.Num		:= 9456;
	xMsg9456.AmmInAdr	:= iAdrAmmBase2MM;
	xMsg9456.AmmOutAdr	:= iAdrMM2AmmBase;

	xMsg9457.Num		:= 9457;
	xMsg9457.AmmInAdr	:= iAdrAmmBase2MM;
	xMsg9457.AmmOutAdr	:= iAdrMM2AmmBase;

	xMsg9458.Num		:= 9458;
	xMsg9458.AmmInAdr	:= iAdrAmmBase2MM;
	xMsg9458.AmmOutAdr	:= iAdrMM2AmmBase;

	xMsg9459.Num		:= 9459;
	xMsg9459.AmmInAdr	:= iAdrAmmBase2MM;
	xMsg9459.AmmOutAdr	:= iAdrMM2AmmBase;

	xMsg9460.Num		:= 9460;
	xMsg9460.AmmInAdr	:= iAdrAmmBase2MM;
	xMsg9460.AmmOutAdr	:= iAdrMM2AmmBase;

	xMsg9461.Num		:= 9461;
	xMsg9461.AmmInAdr	:= iAdrAmmBase2MM;
	xMsg9461.AmmOutAdr	:= iAdrMM2AmmBase;

	xMsg9462.Num		:= 9462;
	xMsg9462.AmmInAdr	:= iAdrAmmBase2MM;
	xMsg9462.AmmOutAdr	:= iAdrMM2AmmBase;

	xMsg9463.Num		:= 9463;
	xMsg9463.AmmInAdr	:= iAdrAmmBase2MM;
	xMsg9463.AmmOutAdr	:= iAdrMM2AmmBase;

	xMsg9464.Num		:= 9464;
	xMsg9464.AmmInAdr	:= iAdrAmmBase2MM;
	xMsg9464.AmmOutAdr	:= iAdrMM2AmmBase;

	xMsg9465.Num		:= 9465;
	xMsg9465.AmmInAdr	:= iAdrAmmBase2MM;
	xMsg9465.AmmOutAdr	:= iAdrMM2AmmBase;

	xMsg9466.Num		:= 9466;
	xMsg9466.AmmInAdr	:= iAdrAmmBase2MM;
	xMsg9466.AmmOutAdr	:= iAdrMM2AmmBase;

	xMsg9467.Num		:= 9467;
	xMsg9467.AmmInAdr	:= iAdrAmmBase2MM;
	xMsg9467.AmmOutAdr	:= iAdrMM2AmmBase;

	xMsg9468.Num		:= 9468;
	xMsg9468.AmmInAdr	:= iAdrAmmBase2MM;
	xMsg9468.AmmOutAdr	:= iAdrMM2AmmBase;

	xMsg9469.Num		:= 9469;
	xMsg9469.AmmInAdr	:= iAdrAmmBase2MM;
	xMsg9469.AmmOutAdr	:= iAdrMM2AmmBase;

	xMsg9470.Num		:= 9470;
	xMsg9470.AmmInAdr	:= iAdrAmmBase2MM;
	xMsg9470.AmmOutAdr	:= iAdrMM2AmmBase;

	xMsg9471.Num		:= 9471;
	xMsg9471.AmmInAdr	:= iAdrAmmBase2MM;
	xMsg9471.AmmOutAdr	:= iAdrMM2AmmBase;

	xMsg9480.Num		:= 9480;
	xMsg9480.AmmInAdr	:= iAdrAmmBase2MM;
	xMsg9480.AmmOutAdr	:= iAdrMM2AmmBase;

	xMsg9481.Num		:= 9481;
	xMsg9481.AmmInAdr	:= iAdrAmmBase2MM;
	xMsg9481.AmmOutAdr	:= iAdrMM2AmmBase;

	xMsg9482.Num		:= 9482;
	xMsg9482.AmmInAdr	:= iAdrAmmBase2MM;
	xMsg9482.AmmOutAdr	:= iAdrMM2AmmBase;

	xMsg9483.Num		:= 9483;
	xMsg9483.AmmInAdr	:= iAdrAmmBase2MM;
	xMsg9483.AmmOutAdr	:= iAdrMM2AmmBase;

	xMsg9484.Num		:= 9484;
	xMsg9484.AmmInAdr	:= iAdrAmmBase2MM;
	xMsg9484.AmmOutAdr	:= iAdrMM2AmmBase;

	xMsg9508.Num		:= 9508;
	xMsg9508.AmmInAdr	:= iAdrAmmBase2MM;
	xMsg9508.AmmOutAdr	:= iAdrMM2AmmBase;

	xMsg9514.Num		:= 9514;
	xMsg9514.AmmInAdr	:= iAdrAmmBase2MM;
	xMsg9514.AmmOutAdr	:= iAdrMM2AmmBase;

	xMsg9515.Num		:= 9515;
	xMsg9515.AmmInAdr	:= iAdrAmmBase2MM;
	xMsg9515.AmmOutAdr	:= iAdrMM2AmmBase;

	xMsg9516.Num		:= 9516;
	xMsg9516.AmmInAdr	:= iAdrAmmBase2MM;
	xMsg9516.AmmOutAdr	:= iAdrMM2AmmBase;

	xMsg9517.Num		:= 9517;
	xMsg9517.AmmInAdr	:= iAdrAmmBase2MM;
	xMsg9517.AmmOutAdr	:= iAdrMM2AmmBase;

	xMsg9518.Num		:= 9518;
	xMsg9518.AmmInAdr	:= iAdrAmmBase2MM;
	xMsg9518.AmmOutAdr	:= iAdrMM2AmmBase;

	xMsg9519.Num		:= 9519;
	xMsg9519.AmmInAdr	:= iAdrAmmBase2MM;
	xMsg9519.AmmOutAdr	:= iAdrMM2AmmBase;

	xMsg9520.Num		:= 9520;
	xMsg9520.AmmInAdr	:= iAdrAmmBase2MM;
	xMsg9520.AmmOutAdr	:= iAdrMM2AmmBase;

	xMsg9521.Num		:= 9521;
	xMsg9521.AmmInAdr	:= iAdrAmmBase2MM;
	xMsg9521.AmmOutAdr	:= iAdrMM2AmmBase;

	xMsg9522.Num		:= 9522;
	xMsg9522.AmmInAdr	:= iAdrAmmBase2MM;
	xMsg9522.AmmOutAdr	:= iAdrMM2AmmBase;

	xMsg9523.Num		:= 9523;
	xMsg9523.AmmInAdr	:= iAdrAmmBase2MM;
	xMsg9523.AmmOutAdr	:= iAdrMM2AmmBase;

	xMsg9524.Num		:= 9524;
	xMsg9524.AmmInAdr	:= iAdrAmmBase2MM;
	xMsg9524.AmmOutAdr	:= iAdrMM2AmmBase;

	xMsg9525.Num		:= 9525;
	xMsg9525.AmmInAdr	:= iAdrAmmBase2MM;
	xMsg9525.AmmOutAdr	:= iAdrMM2AmmBase;

	xMsg9526.Num		:= 9526;
	xMsg9526.AmmInAdr	:= iAdrAmmBase2MM;
	xMsg9526.AmmOutAdr	:= iAdrMM2AmmBase;

	xMsg9527.Num		:= 9527;
	xMsg9527.AmmInAdr	:= iAdrAmmBase2MM;
	xMsg9527.AmmOutAdr	:= iAdrMM2AmmBase;

	xMsg9528.Num		:= 9528;
	xMsg9528.AmmInAdr	:= iAdrAmmBase2MM;
	xMsg9528.AmmOutAdr	:= iAdrMM2AmmBase;

	xMsg9529.Num		:= 9529;
	xMsg9529.AmmInAdr	:= iAdrAmmBase2MM;
	xMsg9529.AmmOutAdr	:= iAdrMM2AmmBase;

	xMsg9530.Num		:= 9530;
	xMsg9530.AmmInAdr	:= iAdrAmmBase2MM;
	xMsg9530.AmmOutAdr	:= iAdrMM2AmmBase;

	xMsg9531.Num		:= 9531;
	xMsg9531.AmmInAdr	:= iAdrAmmBase2MM;
	xMsg9531.AmmOutAdr	:= iAdrMM2AmmBase;

	xMsg9532.Num		:= 9532;
	xMsg9532.AmmInAdr	:= iAdrAmmBase2MM;
	xMsg9532.AmmOutAdr	:= iAdrMM2AmmBase;

	xMsg9533.Num		:= 9533;
	xMsg9533.AmmInAdr	:= iAdrAmmBase2MM;
	xMsg9533.AmmOutAdr	:= iAdrMM2AmmBase;

	xMsg9534.Num		:= 9534;
	xMsg9534.AmmInAdr	:= iAdrAmmBase2MM;
	xMsg9534.AmmOutAdr	:= iAdrMM2AmmBase;

	xMsg9535.Num		:= 9535;
	xMsg9535.AmmInAdr	:= iAdrAmmBase2MM;
	xMsg9535.AmmOutAdr	:= iAdrMM2AmmBase;

	xMsg9536.Num		:= 9536;
	xMsg9536.AmmInAdr	:= iAdrAmmBase2MM;
	xMsg9536.AmmOutAdr	:= iAdrMM2AmmBase;

	xMsg9537.Num		:= 9537;
	xMsg9537.AmmInAdr	:= iAdrAmmBase2MM;
	xMsg9537.AmmOutAdr	:= iAdrMM2AmmBase;

	xMsg9538.Num		:= 9538;
	xMsg9538.AmmInAdr	:= iAdrAmmBase2MM;
	xMsg9538.AmmOutAdr	:= iAdrMM2AmmBase;

	xMsg9539.Num		:= 9539;
	xMsg9539.AmmInAdr	:= iAdrAmmBase2MM;
	xMsg9539.AmmOutAdr	:= iAdrMM2AmmBase;

	xMsg9540.Num		:= 9540;
	xMsg9540.AmmInAdr	:= iAdrAmmBase2MM;
	xMsg9540.AmmOutAdr	:= iAdrMM2AmmBase;

	xMsg9541.Num		:= 9541;
	xMsg9541.AmmInAdr	:= iAdrAmmBase2MM;
	xMsg9541.AmmOutAdr	:= iAdrMM2AmmBase;

	xMsg9542.Num		:= 9542;
	xMsg9542.AmmInAdr	:= iAdrAmmBase2MM;
	xMsg9542.AmmOutAdr	:= iAdrMM2AmmBase;

	xMsg9543.Num		:= 9543;
	xMsg9543.AmmInAdr	:= iAdrAmmBase2MM;
	xMsg9543.AmmOutAdr	:= iAdrMM2AmmBase;

	xMsg9544.Num		:= 9544;
	xMsg9544.AmmInAdr	:= iAdrAmmBase2MM;
	xMsg9544.AmmOutAdr	:= iAdrMM2AmmBase;

	xMsg9545.Num		:= 9545;
	xMsg9545.AmmInAdr	:= iAdrAmmBase2MM;
	xMsg9545.AmmOutAdr	:= iAdrMM2AmmBase;

	xMsg9546.Num		:= 9546;
	xMsg9546.AmmInAdr	:= iAdrAmmBase2MM;
	xMsg9546.AmmOutAdr	:= iAdrMM2AmmBase;

	xMsg9547.Num		:= 9547;
	xMsg9547.AmmInAdr	:= iAdrAmmBase2MM;
	xMsg9547.AmmOutAdr	:= iAdrMM2AmmBase;

	xMsg9548.Num		:= 9548;
	xMsg9548.AmmInAdr	:= iAdrAmmBase2MM;
	xMsg9548.AmmOutAdr	:= iAdrMM2AmmBase;

	xMsg9549.Num		:= 9549;
	xMsg9549.AmmInAdr	:= iAdrAmmBase2MM;
	xMsg9549.AmmOutAdr	:= iAdrMM2AmmBase;

	xMsg9550.Num		:= 9550;
	xMsg9550.AmmInAdr	:= iAdrAmmBase2MM;
	xMsg9550.AmmOutAdr	:= iAdrMM2AmmBase;

	xMsg9551.Num		:= 9551;
	xMsg9551.AmmInAdr	:= iAdrAmmBase2MM;
	xMsg9551.AmmOutAdr	:= iAdrMM2AmmBase;

	xMsg9552.Num		:= 9552;
	xMsg9552.AmmInAdr	:= iAdrAmmBase2MM;
	xMsg9552.AmmOutAdr	:= iAdrMM2AmmBase;

	xMsg9553.Num		:= 9553;
	xMsg9553.AmmInAdr	:= iAdrAmmBase2MM;
	xMsg9553.AmmOutAdr	:= iAdrMM2AmmBase;

	xMsg9554.Num		:= 9554;
	xMsg9554.AmmInAdr	:= iAdrAmmBase2MM;
	xMsg9554.AmmOutAdr	:= iAdrMM2AmmBase;

	xMsg9555.Num		:= 9555;
	xMsg9555.AmmInAdr	:= iAdrAmmBase2MM;
	xMsg9555.AmmOutAdr	:= iAdrMM2AmmBase;

	xMsg9556.Num		:= 9556;
	xMsg9556.AmmInAdr	:= iAdrAmmBase2MM;
	xMsg9556.AmmOutAdr	:= iAdrMM2AmmBase;

	xMsg9562.Num		:= 9562;
	xMsg9562.AmmInAdr	:= iAdrAmmBase2MM;
	xMsg9562.AmmOutAdr	:= iAdrMM2AmmBase;

	xMsg9563.Num		:= 9563;
	xMsg9563.AmmInAdr	:= iAdrAmmBase2MM;
	xMsg9563.AmmOutAdr	:= iAdrMM2AmmBase;

	xMsg9564.Num		:= 9564;
	xMsg9564.AmmInAdr	:= iAdrAmmBase2MM;
	xMsg9564.AmmOutAdr	:= iAdrMM2AmmBase;

	xMsg9565.Num		:= 9565;
	xMsg9565.AmmInAdr	:= iAdrAmmBase2MM;
	xMsg9565.AmmOutAdr	:= iAdrMM2AmmBase;

	xMsg9566.Num		:= 9566;
	xMsg9566.AmmInAdr	:= iAdrAmmBase2MM;
	xMsg9566.AmmOutAdr	:= iAdrMM2AmmBase;

	xMsg9567.Num		:= 9567;
	xMsg9567.AmmInAdr	:= iAdrAmmBase2MM;
	xMsg9567.AmmOutAdr	:= iAdrMM2AmmBase;

	xMsg9568.Num		:= 9568;
	xMsg9568.AmmInAdr	:= iAdrAmmBase2MM;
	xMsg9568.AmmOutAdr	:= iAdrMM2AmmBase;

	xMsg9569.Num		:= 9569;
	xMsg9569.AmmInAdr	:= iAdrAmmBase2MM;
	xMsg9569.AmmOutAdr	:= iAdrMM2AmmBase;

	xMsg9570.Num		:= 9570;
	xMsg9570.AmmInAdr	:= iAdrAmmBase2MM;
	xMsg9570.AmmOutAdr	:= iAdrMM2AmmBase;

	xMsg9571.Num		:= 9571;
	xMsg9571.AmmInAdr	:= iAdrAmmBase2MM;
	xMsg9571.AmmOutAdr	:= iAdrMM2AmmBase;

	xMsg9572.Num		:= 9572;
	xMsg9572.AmmInAdr	:= iAdrAmmBase2MM;
	xMsg9572.AmmOutAdr	:= iAdrMM2AmmBase;

	xMsg9573.Num		:= 9573;
	xMsg9573.AmmInAdr	:= iAdrAmmBase2MM;
	xMsg9573.AmmOutAdr	:= iAdrMM2AmmBase;

	xMsg9574.Num		:= 9574;
	xMsg9574.AmmInAdr	:= iAdrAmmBase2MM;
	xMsg9574.AmmOutAdr	:= iAdrMM2AmmBase;

	xMsg9575.Num		:= 9575;
	xMsg9575.AmmInAdr	:= iAdrAmmBase2MM;
	xMsg9575.AmmOutAdr	:= iAdrMM2AmmBase;

	xMsg9576.Num		:= 9576;
	xMsg9576.AmmInAdr	:= iAdrAmmBase2MM;
	xMsg9576.AmmOutAdr	:= iAdrMM2AmmBase;

	xMsg9577.Num		:= 9577;
	xMsg9577.AmmInAdr	:= iAdrAmmBase2MM;
	xMsg9577.AmmOutAdr	:= iAdrMM2AmmBase;

	xMsg9578.Num		:= 9578;
	xMsg9578.AmmInAdr	:= iAdrAmmBase2MM;
	xMsg9578.AmmOutAdr	:= iAdrMM2AmmBase;

	xMsg9579.Num		:= 9579;
	xMsg9579.AmmInAdr	:= iAdrAmmBase2MM;
	xMsg9579.AmmOutAdr	:= iAdrMM2AmmBase;

	xMsg9580.Num		:= 9580;
	xMsg9580.AmmInAdr	:= iAdrAmmBase2MM;
	xMsg9580.AmmOutAdr	:= iAdrMM2AmmBase;

	xMsg9581.Num		:= 9581;
	xMsg9581.AmmInAdr	:= iAdrAmmBase2MM;
	xMsg9581.AmmOutAdr	:= iAdrMM2AmmBase;

	xMsg9582.Num		:= 9582;
	xMsg9582.AmmInAdr	:= iAdrAmmBase2MM;
	xMsg9582.AmmOutAdr	:= iAdrMM2AmmBase;

	xMsg9583.Num		:= 9583;
	xMsg9583.AmmInAdr	:= iAdrAmmBase2MM;
	xMsg9583.AmmOutAdr	:= iAdrMM2AmmBase;

	xMsg9584.Num		:= 9584;
	xMsg9584.AmmInAdr	:= iAdrAmmBase2MM;
	xMsg9584.AmmOutAdr	:= iAdrMM2AmmBase;

	xMsg9585.Num		:= 9585;
	xMsg9585.AmmInAdr	:= iAdrAmmBase2MM;
	xMsg9585.AmmOutAdr	:= iAdrMM2AmmBase;

	xMsg9586.Num		:= 9586;
	xMsg9586.AmmInAdr	:= iAdrAmmBase2MM;
	xMsg9586.AmmOutAdr	:= iAdrMM2AmmBase;

	xMsg9587.Num		:= 9587;
	xMsg9587.AmmInAdr	:= iAdrAmmBase2MM;
	xMsg9587.AmmOutAdr	:= iAdrMM2AmmBase;

	xMsg9593.Num		:= 9593;
	xMsg9593.AmmInAdr	:= iAdrAmmBase2MM;
	xMsg9593.AmmOutAdr	:= iAdrMM2AmmBase;

	xMsg9597.Num		:= 9597;
	xMsg9597.AmmInAdr	:= iAdrAmmBase2MM;
	xMsg9597.AmmOutAdr	:= iAdrMM2AmmBase;

	xMsg9598.Num		:= 9598;
	xMsg9598.AmmInAdr	:= iAdrAmmBase2MM;
	xMsg9598.AmmOutAdr	:= iAdrMM2AmmBase;

	xMsg9600.Num		:= 9600;
	xMsg9600.AmmInAdr	:= iAdrAmmBase2MM;
	xMsg9600.AmmOutAdr	:= iAdrMM2AmmBase;

	xMsg9627.Num		:= 9627;
	xMsg9627.AmmInAdr	:= iAdrAmmBase2MM;
	xMsg9627.AmmOutAdr	:= iAdrMM2AmmBase;

	xMsg9628.Num		:= 9628;
	xMsg9628.AmmInAdr	:= iAdrAmmBase2MM;
	xMsg9628.AmmOutAdr	:= iAdrMM2AmmBase;

	xMsg9629.Num		:= 9629;
	xMsg9629.AmmInAdr	:= iAdrAmmBase2MM;
	xMsg9629.AmmOutAdr	:= iAdrMM2AmmBase;

	xMsg9630.Num		:= 9630;
	xMsg9630.AmmInAdr	:= iAdrAmmBase2MM;
	xMsg9630.AmmOutAdr	:= iAdrMM2AmmBase;

	xMsg9631.Num		:= 9631;
	xMsg9631.AmmInAdr	:= iAdrAmmBase2MM;
	xMsg9631.AmmOutAdr	:= iAdrMM2AmmBase;

	xMsg9632.Num		:= 9632;
	xMsg9632.AmmInAdr	:= iAdrAmmBase2MM;
	xMsg9632.AmmOutAdr	:= iAdrMM2AmmBase;

	xMsg9633.Num		:= 9633;
	xMsg9633.AmmInAdr	:= iAdrAmmBase2MM;
	xMsg9633.AmmOutAdr	:= iAdrMM2AmmBase;

	xMsg9634.Num		:= 9634;
	xMsg9634.AmmInAdr	:= iAdrAmmBase2MM;
	xMsg9634.AmmOutAdr	:= iAdrMM2AmmBase;

	xMsg9635.Num		:= 9635;
	xMsg9635.AmmInAdr	:= iAdrAmmBase2MM;
	xMsg9635.AmmOutAdr	:= iAdrMM2AmmBase;

	xMsg9636.Num		:= 9636;
	xMsg9636.AmmInAdr	:= iAdrAmmBase2MM;
	xMsg9636.AmmOutAdr	:= iAdrMM2AmmBase;

	xMsg9637.Num		:= 9637;
	xMsg9637.AmmInAdr	:= iAdrAmmBase2MM;
	xMsg9637.AmmOutAdr	:= iAdrMM2AmmBase;

	xMsg9638.Num		:= 9638;
	xMsg9638.AmmInAdr	:= iAdrAmmBase2MM;
	xMsg9638.AmmOutAdr	:= iAdrMM2AmmBase;

	xMsg9639.Num		:= 9639;
	xMsg9639.AmmInAdr	:= iAdrAmmBase2MM;
	xMsg9639.AmmOutAdr	:= iAdrMM2AmmBase;

	xMsg9640.Num		:= 9640;
	xMsg9640.AmmInAdr	:= iAdrAmmBase2MM;
	xMsg9640.AmmOutAdr	:= iAdrMM2AmmBase;

	xMsg9641.Num		:= 9641;
	xMsg9641.AmmInAdr	:= iAdrAmmBase2MM;
	xMsg9641.AmmOutAdr	:= iAdrMM2AmmBase;

	xMsg9642.Num		:= 9642;
	xMsg9642.AmmInAdr	:= iAdrAmmBase2MM;
	xMsg9642.AmmOutAdr	:= iAdrMM2AmmBase;

	xMsg9643.Num		:= 9643;
	xMsg9643.AmmInAdr	:= iAdrAmmBase2MM;
	xMsg9643.AmmOutAdr	:= iAdrMM2AmmBase;

	xMsg9644.Num		:= 9644;
	xMsg9644.AmmInAdr	:= iAdrAmmBase2MM;
	xMsg9644.AmmOutAdr	:= iAdrMM2AmmBase;

	xMsg9645.Num		:= 9645;
	xMsg9645.AmmInAdr	:= iAdrAmmBase2MM;
	xMsg9645.AmmOutAdr	:= iAdrMM2AmmBase;

	xMsg9646.Num		:= 9646;
	xMsg9646.AmmInAdr	:= iAdrAmmBase2MM;
	xMsg9646.AmmOutAdr	:= iAdrMM2AmmBase;

	xMsg9647.Num		:= 9647;
	xMsg9647.AmmInAdr	:= iAdrAmmBase2MM;
	xMsg9647.AmmOutAdr	:= iAdrMM2AmmBase;

	xMsg9648.Num		:= 9648;
	xMsg9648.AmmInAdr	:= iAdrAmmBase2MM;
	xMsg9648.AmmOutAdr	:= iAdrMM2AmmBase;

	xMsg9649.Num		:= 9649;
	xMsg9649.AmmInAdr	:= iAdrAmmBase2MM;
	xMsg9649.AmmOutAdr	:= iAdrMM2AmmBase;

	xMsg9650.Num		:= 9650;
	xMsg9650.AmmInAdr	:= iAdrAmmBase2MM;
	xMsg9650.AmmOutAdr	:= iAdrMM2AmmBase;

	xMsg9651.Num		:= 9651;
	xMsg9651.AmmInAdr	:= iAdrAmmBase2MM;
	xMsg9651.AmmOutAdr	:= iAdrMM2AmmBase;

	xMsg9652.Num		:= 9652;
	xMsg9652.AmmInAdr	:= iAdrAmmBase2MM;
	xMsg9652.AmmOutAdr	:= iAdrMM2AmmBase;

	xMsg9653.Num		:= 9653;
	xMsg9653.AmmInAdr	:= iAdrAmmBase2MM;
	xMsg9653.AmmOutAdr	:= iAdrMM2AmmBase;

	xMsg9654.Num		:= 9654;
	xMsg9654.AmmInAdr	:= iAdrAmmBase2MM;
	xMsg9654.AmmOutAdr	:= iAdrMM2AmmBase;

	xMsg9655.Num		:= 9655;
	xMsg9655.AmmInAdr	:= iAdrAmmBase2MM;
	xMsg9655.AmmOutAdr	:= iAdrMM2AmmBase;

	xMsg9656.Num		:= 9656;
	xMsg9656.AmmInAdr	:= iAdrAmmBase2MM;
	xMsg9656.AmmOutAdr	:= iAdrMM2AmmBase;

	xMsg9657.Num		:= 9657;
	xMsg9657.AmmInAdr	:= iAdrAmmBase2MM;
	xMsg9657.AmmOutAdr	:= iAdrMM2AmmBase;

	xMsg9658.Num		:= 9658;
	xMsg9658.AmmInAdr	:= iAdrAmmBase2MM;
	xMsg9658.AmmOutAdr	:= iAdrMM2AmmBase;

	xMsg9659.Num		:= 9659;
	xMsg9659.AmmInAdr	:= iAdrAmmBase2MM;
	xMsg9659.AmmOutAdr	:= iAdrMM2AmmBase;

	xMsg9660.Num		:= 9660;
	xMsg9660.AmmInAdr	:= iAdrAmmBase2MM;
	xMsg9660.AmmOutAdr	:= iAdrMM2AmmBase;

	xMsg9661.Num		:= 9661;
	xMsg9661.AmmInAdr	:= iAdrAmmBase2MM;
	xMsg9661.AmmOutAdr	:= iAdrMM2AmmBase;

	xMsg9662.Num		:= 9662;
	xMsg9662.AmmInAdr	:= iAdrAmmBase2MM;
	xMsg9662.AmmOutAdr	:= iAdrMM2AmmBase;

	xMsg9663.Num		:= 9663;
	xMsg9663.AmmInAdr	:= iAdrAmmBase2MM;
	xMsg9663.AmmOutAdr	:= iAdrMM2AmmBase;

	xMsg9664.Num		:= 9664;
	xMsg9664.AmmInAdr	:= iAdrAmmBase2MM;
	xMsg9664.AmmOutAdr	:= iAdrMM2AmmBase;

	xMsg9665.Num		:= 9665;
	xMsg9665.AmmInAdr	:= iAdrAmmBase2MM;
	xMsg9665.AmmOutAdr	:= iAdrMM2AmmBase;

	xMsg9666.Num		:= 9666;
	xMsg9666.AmmInAdr	:= iAdrAmmBase2MM;
	xMsg9666.AmmOutAdr	:= iAdrMM2AmmBase;

	xMsg9667.Num		:= 9667;
	xMsg9667.AmmInAdr	:= iAdrAmmBase2MM;
	xMsg9667.AmmOutAdr	:= iAdrMM2AmmBase;

	xMsg9668.Num		:= 9668;
	xMsg9668.AmmInAdr	:= iAdrAmmBase2MM;
	xMsg9668.AmmOutAdr	:= iAdrMM2AmmBase;

	xMsg9669.Num		:= 9669;
	xMsg9669.AmmInAdr	:= iAdrAmmBase2MM;
	xMsg9669.AmmOutAdr	:= iAdrMM2AmmBase;

	xMsg9670.Num		:= 9670;
	xMsg9670.AmmInAdr	:= iAdrAmmBase2MM;
	xMsg9670.AmmOutAdr	:= iAdrMM2AmmBase;

	xMsg9671.Num		:= 9671;
	xMsg9671.AmmInAdr	:= iAdrAmmBase2MM;
	xMsg9671.AmmOutAdr	:= iAdrMM2AmmBase;

	xMsg9672.Num		:= 9672;
	xMsg9672.AmmInAdr	:= iAdrAmmBase2MM;
	xMsg9672.AmmOutAdr	:= iAdrMM2AmmBase;

	xMsg9673.Num		:= 9673;
	xMsg9673.AmmInAdr	:= iAdrAmmBase2MM;
	xMsg9673.AmmOutAdr	:= iAdrMM2AmmBase;

	xMsg9674.Num		:= 9674;
	xMsg9674.AmmInAdr	:= iAdrAmmBase2MM;
	xMsg9674.AmmOutAdr	:= iAdrMM2AmmBase;

	xMsg9675.Num		:= 9675;
	xMsg9675.AmmInAdr	:= iAdrAmmBase2MM;
	xMsg9675.AmmOutAdr	:= iAdrMM2AmmBase;

	xMsg9676.Num		:= 9676;
	xMsg9676.AmmInAdr	:= iAdrAmmBase2MM;
	xMsg9676.AmmOutAdr	:= iAdrMM2AmmBase;

	xMsg9677.Num		:= 9677;
	xMsg9677.AmmInAdr	:= iAdrAmmBase2MM;
	xMsg9677.AmmOutAdr	:= iAdrMM2AmmBase;

	xMsg9678.Num		:= 9678;
	xMsg9678.AmmInAdr	:= iAdrAmmBase2MM;
	xMsg9678.AmmOutAdr	:= iAdrMM2AmmBase;

	xMsg9679.Num		:= 9679;
	xMsg9679.AmmInAdr	:= iAdrAmmBase2MM;
	xMsg9679.AmmOutAdr	:= iAdrMM2AmmBase;

	xMsg9680.Num		:= 9680;
	xMsg9680.AmmInAdr	:= iAdrAmmBase2MM;
	xMsg9680.AmmOutAdr	:= iAdrMM2AmmBase;

	xMsg9681.Num		:= 9681;
	xMsg9681.AmmInAdr	:= iAdrAmmBase2MM;
	xMsg9681.AmmOutAdr	:= iAdrMM2AmmBase;

	xMsg9682.Num		:= 9682;
	xMsg9682.AmmInAdr	:= iAdrAmmBase2MM;
	xMsg9682.AmmOutAdr	:= iAdrMM2AmmBase;

	xMsg9683.Num		:= 9683;
	xMsg9683.AmmInAdr	:= iAdrAmmBase2MM;
	xMsg9683.AmmOutAdr	:= iAdrMM2AmmBase;

	xMsg9684.Num		:= 9684;
	xMsg9684.AmmInAdr	:= iAdrAmmBase2MM;
	xMsg9684.AmmOutAdr	:= iAdrMM2AmmBase;

	xMsg9685.Num		:= 9685;
	xMsg9685.AmmInAdr	:= iAdrAmmBase2MM;
	xMsg9685.AmmOutAdr	:= iAdrMM2AmmBase;

	xMsg9686.Num		:= 9686;
	xMsg9686.AmmInAdr	:= iAdrAmmBase2MM;
	xMsg9686.AmmOutAdr	:= iAdrMM2AmmBase;

	xMsg9687.Num		:= 9687;
	xMsg9687.AmmInAdr	:= iAdrAmmBase2MM;
	xMsg9687.AmmOutAdr	:= iAdrMM2AmmBase;

	xMsg9688.Num		:= 9688;
	xMsg9688.AmmInAdr	:= iAdrAmmBase2MM;
	xMsg9688.AmmOutAdr	:= iAdrMM2AmmBase;

	xMsg9689.Num		:= 9689;
	xMsg9689.AmmInAdr	:= iAdrAmmBase2MM;
	xMsg9689.AmmOutAdr	:= iAdrMM2AmmBase;

	xMsg9690.Num		:= 9690;
	xMsg9690.AmmInAdr	:= iAdrAmmBase2MM;
	xMsg9690.AmmOutAdr	:= iAdrMM2AmmBase;

	xMsg9691.Num		:= 9691;
	xMsg9691.AmmInAdr	:= iAdrAmmBase2MM;
	xMsg9691.AmmOutAdr	:= iAdrMM2AmmBase;

	xMsg9692.Num		:= 9692;
	xMsg9692.AmmInAdr	:= iAdrAmmBase2MM;
	xMsg9692.AmmOutAdr	:= iAdrMM2AmmBase;

	xMsg9693.Num		:= 9693;
	xMsg9693.AmmInAdr	:= iAdrAmmBase2MM;
	xMsg9693.AmmOutAdr	:= iAdrMM2AmmBase;

	xMsg9694.Num		:= 9694;
	xMsg9694.AmmInAdr	:= iAdrAmmBase2MM;
	xMsg9694.AmmOutAdr	:= iAdrMM2AmmBase;

	xMsg9695.Num		:= 9695;
	xMsg9695.AmmInAdr	:= iAdrAmmBase2MM;
	xMsg9695.AmmOutAdr	:= iAdrMM2AmmBase;

	xMsg9696.Num		:= 9696;
	xMsg9696.AmmInAdr	:= iAdrAmmBase2MM;
	xMsg9696.AmmOutAdr	:= iAdrMM2AmmBase;

	xMsg9697.Num		:= 9697;
	xMsg9697.AmmInAdr	:= iAdrAmmBase2MM;
	xMsg9697.AmmOutAdr	:= iAdrMM2AmmBase;

	xMsg9698.Num		:= 9698;
	xMsg9698.AmmInAdr	:= iAdrAmmBase2MM;
	xMsg9698.AmmOutAdr	:= iAdrMM2AmmBase;

	xMsg9699.Num		:= 9699;
	xMsg9699.AmmInAdr	:= iAdrAmmBase2MM;
	xMsg9699.AmmOutAdr	:= iAdrMM2AmmBase;

	xMsg9700.Num		:= 9700;
	xMsg9700.AmmInAdr	:= iAdrAmmBase2MM;
	xMsg9700.AmmOutAdr	:= iAdrMM2AmmBase;

	xMsg9701.Num		:= 9701;
	xMsg9701.AmmInAdr	:= iAdrAmmBase2MM;
	xMsg9701.AmmOutAdr	:= iAdrMM2AmmBase;

	xMsg9702.Num		:= 9702;
	xMsg9702.AmmInAdr	:= iAdrAmmBase2MM;
	xMsg9702.AmmOutAdr	:= iAdrMM2AmmBase;

	xMsg9703.Num		:= 9703;
	xMsg9703.AmmInAdr	:= iAdrAmmBase2MM;
	xMsg9703.AmmOutAdr	:= iAdrMM2AmmBase;

	xMsg9704.Num		:= 9704;
	xMsg9704.AmmInAdr	:= iAdrAmmBase2MM;
	xMsg9704.AmmOutAdr	:= iAdrMM2AmmBase;
END_PROGRAM
```

#### MsgEG.var
```iecst
VAR
	bMsg1056_Set : BOOL := FALSE; (*alarm delayed for one cycle*)
	iAdrAmmBase2MM : UDINT;
	iAdrMM2AmmBase : UDINT;
	iPassLevelReset : INT := 30; (*reset password level - 624 alarms*)
	rP_Ramp_DecGrad : REAL := 1; (*gradient for decrease of power ramp in grid mode [%Pnenn/s] *)
	tiRunOut : TIME := 0; (*Maximum allowed run out time without engine demand*)
	xMsg1026 : Msg; (*FuB*)
	xMsg1031 : Msg; (*FuB*)
	xMsg1056 : Msg; (*FuB*)
	xMsg1168 : Msg; (*FuB*)
	xMsg2190 : Msg; (*FuB*)
	xMsg2191 : Msg; (*FuB*)
	xMsg2192 : Msg; (*FuB*)
	xMsg2193 : Msg; (*FuB*)
	xMsg2194 : Msg; (*FuB*)
	xMsg2195 : Msg; (*FuB*)
	xMsg2196 : Msg; (*FuB*)
	xMsg2197 : Msg; (*FuB*)
	xMsg2198 : Msg; (*FuB*)
	xMsg2199 : Msg; (*FuB*)
	xMsg2200 : Msg; (*FuB*)
	xMsg2227 : Msg; (*FuB*)
	xMsg2228 : Msg; (*FuB*)
	xMsg2229 : Msg; (*FuB*)
	xMsg2230 : Msg; (*FuB*)
	xMsg2232 : Msg; (*FuB*)
	xMsg2270 : Msg; (*FuB*)
	xMsg2285 : Msg; (*FuB*)
	xMsg2286 : Msg; (*FuB*)
	xMsg2300 : Msg; (*FuB*)
	xMsg2362 : Msg; (*FuB*)
	xMsg2383 : Msg; (*FuB*) (*SAFETY PLC*)
	xMsg2384 : Msg; (*FuB*) (*SAFETY PLC*)
	xMsg2385 : Msg; (*FuB*) (*SAFETY PLC*)
	xMsg2386 : Msg; (*FuB*) (*SAFETY PLC*)
	xMsg2387 : Msg; (*FuB*) (*SAFETY PLC*)
	xMsg2388 : Msg; (*FuB*) (*SAFETY PLC*)
	xMsg2389 : Msg; (*FuB*) (*SAFETY PLC*)
	xMsg2390 : Msg; (*FuB*) (*SAFETY PLC*)
	xMsg2391 : Msg; (*FuB*) (*SAFETY PLC*)
	xMsg2392 : Msg; (*FuB*) (*SAFETY PLC*)
	xMsg2393 : Msg; (*FuB*) (*SAFETY PLC*)
	xMsg2394 : Msg; (*FuB*) (*SAFETY PLC*)
	xMsg2395 : Msg; (*FuB*) (*SAFETY PLC*)
	xMsg2396 : Msg; (*FuB*) (*SAFETY PLC*)
	xMsg2397 : Msg; (*FuB*) (*SAFETY PLC*)
	xMsg2398 : Msg; (*FuB*) (*SAFETY PLC*)
	xMsg2542 : Msg; (*FuB*)
	xMsg2544 : Msg; (*FuB*)
	xMsg2552 : Msg; (*FuB*)
	xMsg2553 : Msg; (*FuB*)
	xMsg2561 : Msg; (*FuB*)
	xMsg2790 : Msg; (*FuB*)
	xMsg2794 : Msg; (*FuB*)
	xMsg2804 : Msg; (*FuB*)
	xMsg2805 : Msg; (*FuB*)
	xMsg2806 : Msg; (*FuB*)
	xMsg2807 : Msg; (*FuB*)
	xMsg2822 : Msg; (*FuB*)
	xMsg2904 : Msg; (*FuB*)
	xMsg2905 : Msg; (*FuB*)
	xMsg2909 : Msg; (*FuB*)
	xMsg2958 : Msg; (*FuB*)
	xMsg2959 : Msg; (*FuB*)
	xMsg2981 : Msg; (*FuB*)
	xMsg3368 : Msg; (*FuB*)
	xMsg3378 : Msg; (*FuB*)
	xMsg3396 : Msg; (*FuB*)
	xMsg3449 : Msg; (*FuB*)
	xMsg3559 : Msg; (*FuB*)
	xMsg9038 : Msg; (*FuB*)
	xMsg9217 : Msg; (*FuB*)
	xMsg9218 : Msg; (*FuB*)
	xMsg9219 : Msg; (*FuB*)
	xMsg9408 : Msg; (*FuB*) (*SAFETY PLC*)
	xMsg9409 : Msg; (*FuB*) (*SAFETY PLC*)
	xMsg9410 : Msg; (*FuB*) (*SAFETY PLC*)
	xMsg9411 : Msg; (*FuB*) (*SAFETY PLC*)
	xMsg9412 : Msg; (*FuB*) (*SAFETY PLC*)
	xMsg9413 : Msg; (*FuB*) (*SAFETY PLC*)
	xMsg9414 : Msg; (*FuB*) (*SAFETY PLC*)
	xMsg9415 : Msg; (*FuB*) (*SAFETY PLC*)
	xMsg9416 : Msg; (*FuB*) (*SAFETY PLC*)
	xMsg9417 : Msg; (*FuB*) (*SAFETY PLC*)
	xMsg9418 : Msg; (*FuB*) (*SAFETY PLC*)
	xMsg9419 : Msg; (*FuB*) (*SAFETY PLC*)
	xMsg9420 : Msg; (*FuB*) (*SAFETY PLC*)
	xMsg9421 : Msg; (*FuB*) (*SAFETY PLC*)
	xMsg9422 : Msg; (*FuB*) (*SAFETY PLC*)
	xMsg9423 : Msg; (*FuB*) (*SAFETY PLC*)
	xMsg9424 : Msg; (*FuB*) (*SAFETY PLC*)
	xMsg9425 : Msg; (*FuB*) (*SAFETY PLC*)
	xMsg9426 : Msg; (*FuB*) (*SAFETY PLC*)
	xMsg9427 : Msg; (*FuB*) (*SAFETY PLC*)
	xMsg9428 : Msg; (*FuB*) (*SAFETY PLC*)
	xMsg9429 : Msg; (*FuB*) (*SAFETY PLC*)
	xMsg9430 : Msg; (*FuB*) (*SAFETY PLC*)
	xMsg9431 : Msg; (*FuB*) (*SAFETY PLC*)
	xMsg9433 : Msg; (*FuB*) (*SAFETY PLC*)
	xMsg9434 : Msg; (*FuB*) (*SAFETY PLC*)
	xMsg9437 : Msg; (*FuB*) (*SAFETY PLC*)
	xMsg9438 : Msg; (*FuB*) (*SAFETY PLC*)
	xMsg9439 : Msg; (*FuB*) (*SAFETY PLC*)
	xMsg9440 : Msg; (*FuB*) (*SAFETY PLC*)
	xMsg9441 : Msg; (*FuB*) (*SAFETY PLC*)
	xMsg9442 : Msg; (*FuB*) (*SAFETY PLC*)
	xMsg9443 : Msg; (*FuB*) (*SAFETY PLC*)
	xMsg9444 : Msg; (*FuB*) (*SAFETY PLC*)
	xMsg9445 : Msg; (*FuB*) (*SAFETY PLC*)
	xMsg9446 : Msg; (*FuB*) (*SAFETY PLC*)
	xMsg9447 : Msg; (*FuB*) (*SAFETY PLC*)
	xMsg9448 : Msg; (*FuB*) (*SAFETY PLC*)
	xMsg9449 : Msg; (*FuB*) (*SAFETY PLC*)
	xMsg9450 : Msg; (*FuB*) (*SAFETY PLC*)
	xMsg9451 : Msg; (*FuB*) (*SAFETY PLC*)
	xMsg9452 : Msg; (*FuB*) (*SAFETY PLC*)
	xMsg9453 : Msg; (*FuB*) (*SAFETY PLC*)
	xMsg9454 : Msg; (*FuB*) (*SAFETY PLC*)
	xMsg9455 : Msg; (*FuB*) (*SAFETY PLC*)
	xMsg9456 : Msg; (*FuB*) (*SAFETY PLC*)
	xMsg9457 : Msg; (*FuB*) (*SAFETY PLC*)
	xMsg9458 : Msg; (*FuB*) (*SAFETY PLC*)
	xMsg9459 : Msg; (*FuB*) (*SAFETY PLC*)
	xMsg9460 : Msg; (*FuB*) (*SAFETY PLC*)
	xMsg9461 : Msg; (*FuB*) (*SAFETY PLC*)
	xMsg9462 : Msg; (*FuB*) (*SAFETY PLC*)
	xMsg9463 : Msg; (*FuB*) (*SAFETY PLC*)
	xMsg9464 : Msg; (*FuB*) (*SAFETY PLC*)
	xMsg9465 : Msg; (*FuB*) (*SAFETY PLC*)
	xMsg9466 : Msg; (*FuB*) (*SAFETY PLC*)
	xMsg9467 : Msg; (*FuB*) (*SAFETY PLC*)
	xMsg9468 : Msg; (*FuB*) (*SAFETY PLC*)
	xMsg9469 : Msg; (*FuB*) (*SAFETY PLC*)
	xMsg9470 : Msg; (*FuB*) (*SAFETY PLC*)
	xMsg9471 : Msg; (*FuB*) (*SAFETY PLC*)
	xMsg9480 : Msg; (*FuB*) (*SAFETY PLC*)
	xMsg9481 : Msg; (*FuB*) (*SAFETY PLC*)
	xMsg9482 : Msg; (*FuB*) (*SAFETY PLC*)
	xMsg9483 : Msg; (*FuB*) (*SAFETY PLC*)
	xMsg9484 : Msg; (*FuB*) (*SAFETY PLC*)
	xMsg9508 : Msg; (*FuB*) (*SAFETY PLC*)
	xMsg9514 : Msg; (*FuB*) (*SAFETY PLC*)
	xMsg9515 : Msg; (*FuB*) (*SAFETY PLC*)
	xMsg9516 : Msg; (*FuB*) (*SAFETY PLC*)
	xMsg9517 : Msg; (*FuB*) (*SAFETY PLC*)
	xMsg9518 : Msg; (*FuB*) (*SAFETY PLC*)
	xMsg9519 : Msg; (*FuB*) (*SAFETY PLC*)
	xMsg9520 : Msg; (*FuB*) (*SAFETY PLC*)
	xMsg9521 : Msg; (*FuB*) (*SAFETY PLC*)
	xMsg9522 : Msg; (*FuB*) (*SAFETY PLC*)
	xMsg9523 : Msg; (*FuB*) (*SAFETY PLC*)
	xMsg9524 : Msg; (*FuB*) (*SAFETY PLC*)
	xMsg9525 : Msg; (*FuB*) (*SAFETY PLC*)
	xMsg9526 : Msg; (*FuB*) (*SAFETY PLC*)
	xMsg9527 : Msg; (*FuB*) (*SAFETY PLC*)
	xMsg9528 : Msg; (*FuB*) (*SAFETY PLC*)
	xMsg9529 : Msg; (*FuB*) (*SAFETY PLC*)
	xMsg9530 : Msg; (*FuB*) (*SAFETY PLC*)
	xMsg9531 : Msg; (*FuB*) (*SAFETY PLC*)
	xMsg9532 : Msg; (*FuB*) (*SAFETY PLC*)
	xMsg9533 : Msg; (*FuB*) (*SAFETY PLC*)
	xMsg9534 : Msg; (*FuB*) (*SAFETY PLC*)
	xMsg9535 : Msg; (*FuB*) (*SAFETY PLC*)
	xMsg9536 : Msg; (*FuB*) (*SAFETY PLC*)
	xMsg9537 : Msg; (*FuB*) (*SAFETY PLC*)
	xMsg9538 : Msg; (*FuB*) (*SAFETY PLC*)
	xMsg9539 : Msg; (*FuB*) (*SAFETY PLC*)
	xMsg9540 : Msg; (*FuB*) (*SAFETY PLC*)
	xMsg9541 : Msg; (*FuB*) (*SAFETY PLC*)
	xMsg9542 : Msg; (*FuB*) (*SAFETY PLC*)
	xMsg9543 : Msg; (*FuB*) (*SAFETY PLC*)
	xMsg9544 : Msg; (*FuB*) (*SAFETY PLC*)
	xMsg9545 : Msg; (*FuB*) (*SAFETY PLC*)
	xMsg9546 : Msg; (*FuB*) (*SAFETY PLC*)
	xMsg9547 : Msg; (*FuB*) (*SAFETY PLC*)
	xMsg9548 : Msg; (*FuB*) (*SAFETY PLC*)
	xMsg9549 : Msg; (*FuB*) (*SAFETY PLC*)
	xMsg9550 : Msg; (*FuB*) (*SAFETY PLC*)
	xMsg9551 : Msg; (*FuB*) (*SAFETY PLC*)
	xMsg9552 : Msg; (*FuB*) (*SAFETY PLC*)
	xMsg9553 : Msg; (*FuB*) (*SAFETY PLC*)
	xMsg9554 : Msg; (*FuB*) (*SAFETY PLC*)
	xMsg9555 : Msg; (*FuB*) (*SAFETY PLC*)
	xMsg9556 : Msg; (*FuB*) (*SAFETY PLC*)
	xMsg9562 : Msg; (*FuB*) (*SAFETY PLC*)
	xMsg9563 : Msg; (*FuB*) (*SAFETY PLC*)
	xMsg9564 : Msg; (*FuB*) (*SAFETY PLC*)
	xMsg9565 : Msg; (*FuB*) (*SAFETY PLC*)
	xMsg9566 : Msg; (*FuB*) (*SAFETY PLC*)
	xMsg9567 : Msg; (*FuB*) (*SAFETY PLC*)
	xMsg9568 : Msg; (*FuB*) (*SAFETY PLC*)
	xMsg9569 : Msg; (*FuB*) (*SAFETY PLC*)
	xMsg9570 : Msg; (*FuB*) (*SAFETY PLC*)
	xMsg9571 : Msg; (*FuB*) (*SAFETY PLC*)
	xMsg9572 : Msg; (*FuB*) (*SAFETY PLC*)
	xMsg9573 : Msg; (*FuB*) (*SAFETY PLC*)
	xMsg9574 : Msg; (*FuB*) (*SAFETY PLC*)
	xMsg9575 : Msg; (*FuB*) (*SAFETY PLC*)
	xMsg9576 : Msg; (*FuB*) (*SAFETY PLC*)
	xMsg9577 : Msg; (*FuB*) (*SAFETY PLC*)
	xMsg9578 : Msg; (*FuB*) (*SAFETY PLC*)
	xMsg9579 : Msg; (*FuB*) (*SAFETY PLC*)
	xMsg9580 : Msg; (*FuB*) (*SAFETY PLC*)
	xMsg9581 : Msg; (*FuB*) (*SAFETY PLC*)
	xMsg9582 : Msg; (*FuB*) (*SAFETY PLC*)
	xMsg9583 : Msg; (*FuB*) (*SAFETY PLC*)
	xMsg9584 : Msg; (*FuB*) (*SAFETY PLC*)
	xMsg9585 : Msg; (*FuB*) (*SAFETY PLC*)
	xMsg9586 : Msg; (*FuB*) (*SAFETY PLC*)
	xMsg9587 : Msg; (*FuB*) (*SAFETY PLC*)
	xMsg9593 : Msg; (*FuB*) (*SAFETY PLC*)
	xMsg9597 : Msg; (*FuB*) (*SAFETY PLC*)
	xMsg9598 : Msg; (*FuB*) (*SAFETY PLC*)
	xMsg9600 : Msg; (*FuB*) (*SAFETY PLC*)
	xMsg9627 : Msg; (*FuB*) (*SAFETY PLC*)
	xMsg9628 : Msg; (*FuB*) (*SAFETY PLC*)
	xMsg9629 : Msg; (*FuB*) (*SAFETY PLC*)
	xMsg9630 : Msg; (*FuB*) (*SAFETY PLC*)
	xMsg9631 : Msg; (*FuB*) (*SAFETY PLC*)
	xMsg9632 : Msg; (*FuB*) (*SAFETY PLC*)
	xMsg9633 : Msg; (*FuB*) (*SAFETY PLC*)
	xMsg9634 : Msg; (*FuB*) (*SAFETY PLC*)
	xMsg9635 : Msg; (*FuB*) (*SAFETY PLC*)
	xMsg9636 : Msg; (*FuB*) (*SAFETY PLC*)
	xMsg9637 : Msg; (*FuB*) (*SAFETY PLC*)
	xMsg9638 : Msg; (*FuB*) (*SAFETY PLC*)
	xMsg9639 : Msg; (*FuB*) (*SAFETY PLC*)
	xMsg9640 : Msg; (*FuB*) (*SAFETY PLC*)
	xMsg9641 : Msg; (*FuB*) (*SAFETY PLC*)
	xMsg9642 : Msg; (*FuB*) (*SAFETY PLC*)
	xMsg9643 : Msg; (*FuB*) (*SAFETY PLC*)
	xMsg9644 : Msg; (*FuB*) (*SAFETY PLC*)
	xMsg9645 : Msg; (*FuB*) (*SAFETY PLC*)
	xMsg9646 : Msg; (*FuB*) (*SAFETY PLC*)
	xMsg9647 : Msg; (*FuB*) (*SAFETY PLC*)
	xMsg9648 : Msg; (*FuB*) (*SAFETY PLC*)
	xMsg9649 : Msg; (*FuB*) (*SAFETY PLC*)
	xMsg9650 : Msg; (*FuB*) (*SAFETY PLC*)
	xMsg9651 : Msg; (*FuB*) (*SAFETY PLC*)
	xMsg9652 : Msg; (*FuB*) (*SAFETY PLC*)
	xMsg9653 : Msg; (*FuB*) (*SAFETY PLC*)
	xMsg9654 : Msg; (*FuB*) (*SAFETY PLC*)
	xMsg9655 : Msg; (*FuB*) (*SAFETY PLC*)
	xMsg9656 : Msg; (*FuB*) (*SAFETY PLC*)
	xMsg9657 : Msg; (*FuB*) (*SAFETY PLC*)
	xMsg9658 : Msg; (*FuB*) (*SAFETY PLC*)
	xMsg9659 : Msg; (*FuB*) (*SAFETY PLC*)
	xMsg9660 : Msg; (*FuB*) (*SAFETY PLC*)
	xMsg9661 : Msg; (*FuB*) (*SAFETY PLC*)
	xMsg9662 : Msg; (*FuB*) (*SAFETY PLC*)
	xMsg9663 : Msg; (*FuB*) (*SAFETY PLC*)
	xMsg9664 : Msg; (*FuB*) (*SAFETY PLC*)
	xMsg9665 : Msg; (*FuB*) (*SAFETY PLC*)
	xMsg9666 : Msg; (*FuB*) (*SAFETY PLC*)
	xMsg9667 : Msg; (*FuB*) (*SAFETY PLC*)
	xMsg9668 : Msg; (*FuB*) (*SAFETY PLC*)
	xMsg9669 : Msg; (*FuB*) (*SAFETY PLC*)
	xMsg9670 : Msg; (*FuB*) (*SAFETY PLC*)
	xMsg9671 : Msg; (*FuB*) (*SAFETY PLC*)
	xMsg9672 : Msg; (*FuB*) (*SAFETY PLC*)
	xMsg9673 : Msg; (*FuB*) (*SAFETY PLC*)
	xMsg9674 : Msg; (*FuB*) (*SAFETY PLC*)
	xMsg9675 : Msg; (*FuB*) (*SAFETY PLC*)
	xMsg9676 : Msg; (*FuB*) (*SAFETY PLC*)
	xMsg9677 : Msg; (*FuB*) (*SAFETY PLC*)
	xMsg9678 : Msg; (*FuB*) (*SAFETY PLC*)
	xMsg9679 : Msg; (*FuB*) (*SAFETY PLC*)
	xMsg9680 : Msg; (*FuB*) (*SAFETY PLC*)
	xMsg9681 : Msg; (*FuB*) (*SAFETY PLC*)
	xMsg9682 : Msg; (*FuB*) (*SAFETY PLC*)
	xMsg9683 : Msg; (*FuB*) (*SAFETY PLC*)
	xMsg9684 : Msg; (*FuB*) (*SAFETY PLC*)
	xMsg9685 : Msg; (*FuB*) (*SAFETY PLC*)
	xMsg9686 : Msg; (*FuB*) (*SAFETY PLC*)
	xMsg9687 : Msg; (*FuB*) (*SAFETY PLC*)
	xMsg9688 : Msg; (*FuB*) (*SAFETY PLC*)
	xMsg9689 : Msg; (*FuB*) (*SAFETY PLC*)
	xMsg9690 : Msg; (*FuB*) (*SAFETY PLC*)
	xMsg9691 : Msg; (*FuB*) (*SAFETY PLC*)
	xMsg9692 : Msg; (*FuB*) (*SAFETY PLC*)
	xMsg9693 : Msg; (*FuB*) (*SAFETY PLC*)
	xMsg9694 : Msg; (*FuB*) (*SAFETY PLC*)
	xMsg9695 : Msg; (*FuB*) (*SAFETY PLC*)
	xMsg9696 : Msg; (*FuB*) (*SAFETY PLC*)
	xMsg9697 : Msg; (*FuB*) (*SAFETY PLC*)
	xMsg9698 : Msg; (*FuB*) (*SAFETY PLC*)
	xMsg9699 : Msg; (*FuB*) (*SAFETY PLC*)
	xMsg9700 : Msg; (*FuB*) (*SAFETY PLC*)
	xMsg9701 : Msg; (*FuB*) (*SAFETY PLC*)
	xMsg9702 : Msg; (*FuB*) (*SAFETY PLC*)
	xMsg9703 : Msg; (*FuB*) (*SAFETY PLC*)
	xMsg9704 : Msg; (*FuB*) (*SAFETY PLC*)
	xTOF_Calib_Ok : TOF := (0); (*FuB*)
	xTON_1026_A : TON := (0); (*FuB*)
	xTON_1026_B : TON := (0); (*FuB*)
	xTON_1026_C : TON := (0); (*FuB*)
END_VAR
```

### Program Logical/EngineGeneral/ParEG (IEC, version 4.06.0) - + save parameters

- perm_par.st (not readable text: treated as protected, skipped)

#### perm_par.var
```iecst
VAR
	tParaIntern : ParaHandler_typ; (*Connector type to perm_par*)
	tMM2ParaBase_ReadBack : MM2ParaBase_type; (*INTERNAL! V4.06 new readback structure for information from previous tasks*)
	bWriteDataObj : BOOL; (* TRUE=write data object module *)
	bDataObjLenErr : BOOL; (*Error occured in permem: data module size missmatch*)
	bCreateDataObj : BOOL; (* TRUE=create new data object *)
	bWriteOnce : BOOL; (* write permanent memory once *)
	DatObjCreate_01 : DatObjCreate; (* data object create *)
	DatObjInfoBak_02 : DatObjInfo; (* data object info *)
	DatObjDelete_01 : DatObjDelete; (* data object delete *)
	DatObjRead_01 : DatObjRead; (* data object read *)
	DatObjRead_02 : DatObjRead; (* manual initiated data object read *)
	DatObjWrite_01 : DatObjWrite; (* data object write *)
	DatObjDelete_02 : DatObjDelete; (* data object delete *)
	DatObjDelete_11 : DatObjDelete; (*Delete Backup File*)
	DatObjInfo_01 : DatObjInfo; (* data object info *)
	DatObjInfo_02 : DatObjInfo; (* data object info *)
	szModuleName : STRING[35]; (* module name of object *)
	szModuleNameBackup : STRING[35]; (* module name of posiibly created backup object *)
	DatObjCopy_01 : DatObjCopy;
	bCopyDataObj : BOOL;
	TON_WarnDelay : TON;
	TON_WritePMEM : TON; (* delay write permanent memory *)
	ulPMPointer : UDINT; (* adress of actual checksum value *)
	ulChecksum : UDINT; (* parameter checksum value *)
	pm_len : UDINT; (* permanent value lenght *)
	ulChecksumOld : UDINT; (* last vlaue of parameter checksum *)
	ulChkValue : UDINT; (* actual value of parameter pointer *)
	pm_id : UDINT; (* permanent value identifier *)
	pm_p : UDINT; (* permanent value pointer *)
	DatObjInfo_META : DatObjInfo;
	DatObjRead_META : DatObjRead;
	szMetaDataRaw : STRING[2000];
	szMetaData : ARRAY[0..4] OF STRING[35];
	szMetaDataVis : ARRAY[0..3] OF STRING[35];
	ssIndex : INT;
	ssCount : INT;
	ucMetaDataRaw : ARRAY[0..2000] OF USINT;
	ssCount2 : INT;
	szMetaDataFile : STRING[10];
	szText1 : STRING[20];
	pv_adr_IN_XX_tPB2MM : UDINT;
	pv_lng : UDINT;
	pv_lng_IN_XX_tPB2MM : UDINT;
	pv_lng_OUT_XX_tPB2MM : UDINT;
	szText2 : STRING[20];
	pv_adr_OUT_XX_tXX2PB : UDINT;
END_VAR
VAR CONSTANT
	ERR_NOERROR : UINT := 0;
END_VAR
VAR
	usPMWriteCnt : UINT;
	pm_Error : UDINT; (* permanent value error *) (* Deleted: pm : ParaMem_typ; permanent memory tags mathias, 22.8.11*)
	fun_Error : UDINT := 0; (*state > 0 = function error*)
	xLocalParaCheck : ParaCheckFUB; (*local function instance to check parameter values*)
	TON_ParaSetupOk : TON;
	bParaCheckSystemOk : BOOL;
	iDebug_ParaOkChecked : UDINT;
	bRestoreBackupDataObj : BOOL := FALSE;
	bRestoreDataObjContent : BOOL := FALSE;
	pm_id_backup : UDINT;
	pm_p_Backup : UDINT;
	DatObjCopy_02 : DatObjCopy;
	bDeleteBackupDataObj : BOOL := FALSE; (*Command to delete backup data module file on purpose*)
	bDebugPara : ARRAY[0..5] OF BOOL;
	ssIndex2 : INT;
	ssIndex3 : INT;
	ssIndex4 : INT;
	ssIndexVis : INT;
	szText : STRING[40];
	pv_adr_Para : UDINT;
	szParaSnippet : ARRAY[0..5] OF STRING[150];
	szParaIndex : STRING[10];
	slValue : DINT;
	iModuleDLD_ResetCount : INT;
	bDownloadDetected : BOOL;
	bFlagParaStructCopyWorking : BOOL; (*true, if cyclic para copying is active, 1 false cycle at every copy *)
	bStoreInitParaInDataObj : BOOL := FALSE;
	bTestflag : BOOL;
	bReadOutMETA_Once : BOOL;
	tParaCheck_iPvAdress : ARRAY[0..5] OF UDINT;
	tParaCheck_iPvLengt : ARRAY[0..5] OF UDINT;
	tParaCheck_rPvValue : ARRAY[0..5] OF REAL;
	tParaCheck_rRangeMIN : ARRAY[0..5] OF REAL;
	tParaCheck_rRangeMAX : ARRAY[0..5] OF REAL;
	tParaCheck_szPvName : ARRAY[0..5] OF STRING[35];
	ssFormatDetected : INT;
	szMetaDataPart : STRING[150];
	szFullTaskName : STRING[35];
	szFullMetaModuleName : STRING[35];
	debugLen : INT;
	debugSize : INT := 0;
	strcat_adr1 : UDINT;
	strcat_adr2 : UDINT;
	ssIndexTN : INT;
	bAlternate : BOOL;
	n : INT;
	iAlternateChecksum : DINT;
	iAlternateChecksumOld : DINT;
	ulDebugChkValue : ARRAY[0..999] OF UDINT;
	Adr1 : UDINT;
	Adr2 : UDINT;
	usPMWriteCntStepsize : UINT := 1; (*different step sizes to help debug*)
	usPMWriteCntXOR : UINT;
	usPMWriteCntAltSum : UINT;
	ulAdrPM : UDINT;
	usChkValuePM : USINT;
	ulAdrPara : UDINT;
	ulPara_len : UDINT;
	usChkValuePara : USINT;
	iDebugCountPMDifferences : DINT := 0;
	bEngineRunDetected : BOOL; (*detection status bit autocommand 100 /101  for engine run state*)
	ucMetaDataDebugInfoLine : ARRAY[0..24] OF STRING[80];
	ssIndexMand : INT := 0;
	szMetaDataMand : STRING[35];
	iMyErrorInfo_Autoreset : DINT; (*internal autoreset counter*)
	ssIndex_Version : INT; (*internal*)
	ssIndex_BU : INT; (*internal*)
	ssIndex_BU2 : INT; (*internal*)
END_VAR
```

### Program Logical/EngineGeneral/VibMonEG (IEC, version 4.11.2) - Vibration monitoring eng & gen

#### VibMonEGCyclic.st - Init, cyclic, exit code
```iecst
(*******************************************************************************
VibMonEG: Vigration monitoring engine / generator (cyclic)

This code is confidential AND proprietary to the INNIO Company.
It may NOT be used in any form, or reproduced in any manner, without the express
written permission of the INNIO Company.
Copyright, INNIO Company, 2021

- monitoring of vibration values incl. frequency bands
- determine max velocity and frequencay at maximum

Customized modifications: -
------------------------

History:
-------
V4.11	25-05-2021	Weitzer, 	generated

Instructions FOR use:
--------------------
Sensor 1: Generator horizontal
Sensor 2: Generator vetical
Sensor 3: Engine horizontal
Sensor 4: Engine vetical

Outstandings:
------------

*******************************************************************************)

PROGRAM _CYCLIC

	(* code is only executed if function is activated by parameter and if system has completed the start up *)
	IF Para.bVibSens_Act AND IN_EG.tPB2MM.bSys_Run THEN

		(* mapping of data points from 4 vibration sensors *)
		FOR usCount := 0 TO 3 DO

			(* check if vibraton sensore wire break detected and engine speed is below start limit *)
			IF bVibSens_BrokenWire[usCount+1] OR IN_EG.rN_EngAct < Para.rN_EngStart_LimHi THEN
				(* vibration sensor live RMS values [mm/s]*)
				MM2VIS.rVel_VibSens[usCount+1] := 0;
				(* vibration sensor live frequency band [mm/s] *)
				MM2VIS.rVel_VibSens_Band1[usCount+1] := 0;
				MM2VIS.rVel_VibSens_Band2[usCount+1] := 0;
				MM2VIS.rVel_VibSens_Band3[usCount+1] := 0;
				MM2VIS.rVel_VibSens_Band4[usCount+1] := 0;
				MM2VIS.rVel_VibSens_Band5[usCount+1] := 0;
				MM2VIS.rVel_VibSens_Band6[usCount+1] := 0;
				MM2VIS.rVel_VibSens_Band7[usCount+1] := 0;
				MM2VIS.rVel_VibSens_Band8[usCount+1] := 0;
				(* vibration sensor max values *)
				MM2VIS.rVel_VibSens_Max[usCount+1] := 0;
				MM2VIS.rF_VibSens_Max[usCount+1]   := 0;
			(* check if no vibraton sensore overflow detected *)
			ELSIF NOT bVibSens_Overflow[usCount+1] THEN
				(* vibration sensor live RMS values [mm/s]*)
				MM2VIS.rVel_VibSens[usCount+1] := rVel_VibSens[usCount+1];					(* mapping directly from IO mapping, no HALIO used for vibration mesarurement *)
				(* vibration sensor live frequency band [mm/s] *)
				MM2VIS.rVel_VibSens_Band1[usCount+1] := rVel_VibSens_Band[usCount*8+1];		(* mapping directly from IO mapping, no HALIO used for vibration mesarurement *)
				MM2VIS.rVel_VibSens_Band2[usCount+1] := rVel_VibSens_Band[usCount*8+2];		(* mapping directly from IO mapping, no HALIO used for vibration mesarurement *)
				MM2VIS.rVel_VibSens_Band3[usCount+1] := rVel_VibSens_Band[usCount*8+3];		(* mapping directly from IO mapping, no HALIO used for vibration mesarurement *)
				MM2VIS.rVel_VibSens_Band4[usCount+1] := rVel_VibSens_Band[usCount*8+4];		(* mapping directly from IO mapping, no HALIO used for vibration mesarurement *)
				MM2VIS.rVel_VibSens_Band5[usCount+1] := rVel_VibSens_Band[usCount*8+5];		(* mapping directly from IO mapping, no HALIO used for vibration mesarurement *)
				MM2VIS.rVel_VibSens_Band6[usCount+1] := rVel_VibSens_Band[usCount*8+6];		(* mapping directly from IO mapping, no HALIO used for vibration mesarurement *)
				MM2VIS.rVel_VibSens_Band7[usCount+1] := rVel_VibSens_Band[usCount*8+7];		(* mapping directly from IO mapping, no HALIO used for vibration mesarurement *)
				MM2VIS.rVel_VibSens_Band8[usCount+1] := rVel_VibSens_Band[usCount*8+8];		(* mapping directly from IO mapping, no HALIO used for vibration mesarurement *)
			END_IF;

		END_FOR;

		(* read buffer data *)

		(* generate time interval for reading buffer *)
		xTON_ReadCycle(IN := NOT xTON_ReadCycle.Q, PT :=  tiCM4810_ReadBuffer);

		(* generate start reading trigger *)
		IF IN_EG.tEng_Run.Do AND stpCM4810 = stpWaitStart AND xTON_ReadCycle.Q THEN
			iNum_VibSens := iNum_VibSens + 1;
			IF iNum_VibSens > 4 THEN
				iNum_VibSens := 1;
			END_IF;
			bStartBufferUpload 					   := TRUE;
			xCM4810.paramBufferUpload.moduleBuffer := 66 + (iNum_VibSens-1) * 4;
		END_IF;

		(* state engine to read of data buffer *)

		CASE stpCM4810 OF
			//---------------------------------------------
			// wait for init done
			//---------------------------------------------
			stpInitDone:
				xCM4810.requestBufferLock := FALSE;
				xCM4810.uploadBuffer	  := FALSE;
				IF xCM4810.initDone AND xCM4810.moduleCfgUploadDone THEN
					stpCM4810 := stpWaitStart;
				END_IF;

			//---------------------------------------------
			// wait for start uplaod buffer
			//---------------------------------------------
			stpWaitStart:
				xCM4810.requestBufferLock := FALSE;
				xCM4810.uploadBuffer	  := FALSE;
				(* wait for start *)
				IF bStartBufferUpload THEN
					stpCM4810 := stpReqLockBuffer;
				END_IF;

			//---------------------------------------------
			// request lock buffer and wait until valid
			//---------------------------------------------
			stpReqLockBuffer:
				xCM4810.requestBufferLock := TRUE;
				bStartBufferUpload		  := FALSE; (* reset command start *)
				IF xCM4810.bufferLockValid THEN
					xCM4810.uploadBuffer := TRUE;
					stpCM4810			 := stpUploadBuffer;
				END_IF;

			//---------------------------------------------
			// upload buffer
			//---------------------------------------------
			stpUploadBuffer:
				IF xCM4810.bufferUploadDone THEN
					stpCM4810 := stpReqUnlockBuffer;
				END_IF;
				IF xCM4810.status <> ERR_FUB_BUSY AND xCM4810.status <> ERR_OK THEN
					stpCM4810 := stpError;
				END_IF

			//---------------------------------------------
			// unlock buffer and wait until valid
			//---------------------------------------------
			stpReqUnlockBuffer:
				xCM4810.requestBufferLock := FALSE;
				xCM4810.uploadBuffer	  := FALSE;
				IF NOT xCM4810.bufferLockValid THEN
					bGetFrequencyMax := TRUE;
					stpCM4810		 := stpWaitStart;
				END_IF;

			//---------------------------------------------
			// error
			//---------------------------------------------
			stpError:
			// no action!

		END_CASE;

		xCM4810.paramMain.pModulePath			  := ADR(sCM4810Addr);
		xCM4810.paramBufferUpload.pArrayXaxis	  := ADR(rData_x_Axis);
		xCM4810.paramBufferUpload.pArrayYaxis	  := ADR(rData_y_Axis);

		xCM4810(); (* call FUB exactly once per cycle *)

		(* get value & frequency max *)

		IF bGetFrequencyMax THEN

			MM2VIS.rF_VibSens_Max[iNum_VibSens]   := 0.0;		(* reset x(y max) max *)
			rVel_y_Axis_Max := 0.0;										(* reset y max *)
			usMaxIndex := 0;
			FOR usCount := 1 TO AxisArrayMaxIndex DO
				(* Upper limit for max value search at 500 Hz *)
				IF rData_x_Axis[usCount] > 500.0 THEN
					EXIT;
				END_IF
				(*find max signal value *)
				IF rData_y_Axis[usCount] > rVel_y_Axis_Max THEN
					rVel_y_Axis_Max := rData_y_Axis[usCount];		(* max virbration value *)
					MM2VIS.rF_VibSens_Max[iNum_VibSens]   := rData_x_Axis[usCount];		(* frequency at max virbration value *)
					usMaxIndex := usCount;
				END_IF
			END_FOR;

			(* correction of buffer value *)
			IF usMaxIndex > 1 AND usMaxIndex < (AxisArrayMaxIndex-2) THEN
				MM2VIS.rVel_VibSens_Max[iNum_VibSens] := 2.0/SQRT(3.0/2.0)*SQRT(0.5*(EXPT(rData_y_Axis[usMaxIndex-2],2)+EXPT(rData_y_Axis[usMaxIndex-1],2)+EXPT(rData_y_Axis[usMaxIndex],2)+EXPT(rData_y_Axis[usMaxIndex+1],2)+EXPT(rData_y_Axis[usMaxIndex+2],2)));
			ELSE
				MM2VIS.rVel_VibSens_Max[iNum_VibSens] := 0.0;
			END_IF;

			bGetFrequencyMax := FALSE;
		END_IF;

		(* calculate and display center frequency at the HMI *)

		MM2VIS.rF_VibSens_CenterBand1 := Para.rN_EngNom/60.0*Para.rIdx_VibSens_BandOrder1;
		MM2VIS.rF_VibSens_CenterBand2 := Para.rN_EngNom/60.0*Para.rIdx_VibSens_BandOrder2;
		MM2VIS.rF_VibSens_CenterBand3 := Para.rN_EngNom/60.0*Para.rIdx_VibSens_BandOrder3;
		MM2VIS.rF_VibSens_CenterBand4 := Para.rN_EngNom/60.0*Para.rIdx_VibSens_BandOrder4;
		MM2VIS.rF_VibSens_CenterBand5 := Para.rN_EngNom/60.0*Para.rIdx_VibSens_BandOrder5;
		MM2VIS.rF_VibSens_CenterBand6 := Para.rN_EngNom/60.0*Para.rIdx_VibSens_BandOrder6;
		MM2VIS.rF_VibSens_CenterBand7 := Para.rN_EngNom/60.0*Para.rIdx_VibSens_BandOrder7;
		MM2VIS.rF_VibSens_CenterBand8 := Para.rN_EngNom/60.0*Para.rIdx_VibSens_BandOrder8;

		(* check if band upper and lower frequency limit has to be set *)

		IF NOT bWrite THEN

			IF ucWriteBandCnt = 0 THEN

				IF Para.rIdx_VibSens_BandWidth <> rIdx_VibSens_BandWidtOld THEN
					rIdx_VibSens_BandWidtOld := Para.rIdx_VibSens_BandWidth;
					rCenterBandOld1			 := 0.0;
					rCenterBandOld2			 := 0.0;
					rCenterBandOld3			 := 0.0;
					rCenterBandOld4			 := 0.0;
					rCenterBandOld5			 := 0.0;
					rCenterBandOld6			 := 0.0;
					rCenterBandOld7			 := 0.0;
					rCenterBandOld8			 := 0.0;
				ELSIF MM2VIS.rF_VibSens_CenterBand1 <> rCenterBandOld1 THEN
					rCenterBandOld1 := MM2VIS.rF_VibSens_CenterBand1;
					ucWriteBandCnt  := 1;
				ELSIF MM2VIS.rF_VibSens_CenterBand2 <> rCenterBandOld2 THEN
					rCenterBandOld2 := MM2VIS.rF_VibSens_CenterBand2;
					ucWriteBandCnt  := 9;
				ELSIF MM2VIS.rF_VibSens_CenterBand3 <> rCenterBandOld3 THEN
					rCenterBandOld3 := MM2VIS.rF_VibSens_CenterBand3;
					ucWriteBandCnt  := 17;
				ELSIF MM2VIS.rF_VibSens_CenterBand4 <> rCenterBandOld4 THEN
					rCenterBandOld4 := MM2VIS.rF_VibSens_CenterBand4;
					ucWriteBandCnt  := 25;
				ELSIF MM2VIS.rF_VibSens_CenterBand5 <> rCenterBandOld5 THEN
					rCenterBandOld5 := MM2VIS.rF_VibSens_CenterBand5;
					ucWriteBandCnt  := 33;
				ELSIF MM2VIS.rF_VibSens_CenterBand6 <> rCenterBandOld6 THEN
					rCenterBandOld6 := MM2VIS.rF_VibSens_CenterBand6;
					ucWriteBandCnt  := 41;
				ELSIF MM2VIS.rF_VibSens_CenterBand7 <> rCenterBandOld7 THEN
					rCenterBandOld7 := MM2VIS.rF_VibSens_CenterBand7;
					ucWriteBandCnt  := 49;
				ELSIF MM2VIS.rF_VibSens_CenterBand8 <> rCenterBandOld8 THEN
					rCenterBandOld8 := MM2VIS.rF_VibSens_CenterBand8;
					ucWriteBandCnt  := 57;
				END_IF;

			END_IF;

			(* writing of the single band limit registers *)
			CASE ucWriteBandCnt OF

				(* Band 1 - Sensor 1 *)
				1:  bWrite		 		 := TRUE;
					szWriteConfig		 := 'FrequencyBand01LowerFrequency';
					xAsIOAccWrite1.value := LIMIT(1,REAL_TO_UDINT(4.0*(MM2VIS.rF_VibSens_CenterBand1 - Para.rIdx_VibSens_BandWidth/2)),40000);
					ucWriteBandCnt		 := 2;
				2:  bWrite		 		 := TRUE;
					szWriteConfig		 := 'FrequencyBand01UpperFrequency';
					xAsIOAccWrite1.value := LIMIT(1,REAL_TO_UDINT(4.0*(MM2VIS.rF_VibSens_CenterBand1 + Para.rIdx_VibSens_BandWidth/2)),40000);
					ucWriteBandCnt		 := 3;
				(* Band 1 - Sensor 2 *)
				3:  bWrite		 		 := TRUE;
					szWriteConfig		 := 'FrequencyBand09LowerFrequency';
					xAsIOAccWrite1.value := LIMIT(1,REAL_TO_UDINT(4.0*(MM2VIS.rF_VibSens_CenterBand1 - Para.rIdx_VibSens_BandWidth/2)),40000);
					ucWriteBandCnt		 := 4;
				4:  bWrite		 		 := TRUE;
					szWriteConfig		 := 'FrequencyBand09UpperFrequency';
					xAsIOAccWrite1.value := LIMIT(1,REAL_TO_UDINT(4.0*(MM2VIS.rF_VibSens_CenterBand1 + Para.rIdx_VibSens_BandWidth/2)),40000);
					ucWriteBandCnt		 := 5;
				(* Band 1 - Sensor 3 *)
				5:  bWrite		 		 := TRUE;
					szWriteConfig		 := 'FrequencyBand17LowerFrequency';
					xAsIOAccWrite1.value := LIMIT(1,REAL_TO_UDINT(4.0*(MM2VIS.rF_VibSens_CenterBand1 - Para.rIdx_VibSens_BandWidth/2)),40000);
					ucWriteBandCnt		 := 6;
				6:  bWrite		 		 := TRUE;
					szWriteConfig		 := 'FrequencyBand17UpperFrequency';
					xAsIOAccWrite1.value := LIMIT(1,REAL_TO_UDINT(4.0*(MM2VIS.rF_VibSens_CenterBand1 + Para.rIdx_VibSens_BandWidth/2)),40000);
					ucWriteBandCnt		 := 7;
				(* Band 1 - Sensor 4 *)
				7:  bWrite		 		 := TRUE;
					szWriteConfig		 := 'FrequencyBand25LowerFrequency';
					xAsIOAccWrite1.value := LIMIT(1,REAL_TO_UDINT(4.0*(MM2VIS.rF_VibSens_CenterBand1 - Para.rIdx_VibSens_BandWidth/2)),40000);
					ucWriteBandCnt		 := 8;
				8:  bWrite		 		 := TRUE;
					szWriteConfig		 := 'FrequencyBand25UpperFrequency';
					xAsIOAccWrite1.value := LIMIT(1,REAL_TO_UDINT(4.0*(MM2VIS.rF_VibSens_CenterBand1 + Para.rIdx_VibSens_BandWidth/2)),40000);
					ucWriteBandCnt		 := 0;

					(* Band 2 - Sensor 1 *)
				9:  bWrite		 		 := TRUE;
					szWriteConfig		 := 'FrequencyBand02LowerFrequency';
					xAsIOAccWrite1.value := LIMIT(1,REAL_TO_UDINT(4.0*(MM2VIS.rF_VibSens_CenterBand2 - Para.rIdx_VibSens_BandWidth/2)),40000);
					ucWriteBandCnt		 := 10;
				10: bWrite		 		 := TRUE;
					szWriteConfig		 := 'FrequencyBand02UpperFrequency';
					xAsIOAccWrite1.value := LIMIT(1,REAL_TO_UDINT(4.0*(MM2VIS.rF_VibSens_CenterBand2 + Para.rIdx_VibSens_BandWidth/2)),40000);
					ucWriteBandCnt		 := 11;
					(* Band 2 - Sensor 2 *)
				11: bWrite		 		 := TRUE;
					szWriteConfig		 := 'FrequencyBand10LowerFrequency';
					xAsIOAccWrite1.value := LIMIT(1,REAL_TO_UDINT(4.0*(MM2VIS.rF_VibSens_CenterBand2 - Para.rIdx_VibSens_BandWidth/2)),40000);
					ucWriteBandCnt		 := 12;
				12: bWrite		 		 := TRUE;
					szWriteConfig		 := 'FrequencyBand10UpperFrequency';
					xAsIOAccWrite1.value := LIMIT(1,REAL_TO_UDINT(4.0*(MM2VIS.rF_VibSens_CenterBand2 + Para.rIdx_VibSens_BandWidth/2)),40000);
					ucWriteBandCnt		 := 13;
					(* Band 2 - Sensor 3 *)
				13: bWrite		 		 := TRUE;
					szWriteConfig		 := 'FrequencyBand18LowerFrequency';
					xAsIOAccWrite1.value := LIMIT(1,REAL_TO_UDINT(4.0*(MM2VIS.rF_VibSens_CenterBand2 - Para.rIdx_VibSens_BandWidth/2)),40000);
					ucWriteBandCnt		 := 14;
				14: bWrite		 		 := TRUE;
					szWriteConfig		 := 'FrequencyBand18UpperFrequency';
					xAsIOAccWrite1.value := LIMIT(1,REAL_TO_UDINT(4.0*(MM2VIS.rF_VibSens_CenterBand2 + Para.rIdx_VibSens_BandWidth/2)),40000);
					ucWriteBandCnt		 := 15;
					(* Band 2 - Sensor 4 *)
				15: bWrite		 		 := TRUE;
					szWriteConfig		 := 'FrequencyBand26LowerFrequency';
					xAsIOAccWrite1.value := LIMIT(1,REAL_TO_UDINT(4.0*(MM2VIS.rF_VibSens_CenterBand2 - Para.rIdx_VibSens_BandWidth/2)),40000);
					ucWriteBandCnt		 := 16;
				16: bWrite		 		 := TRUE;
					szWriteConfig		 := 'FrequencyBand26UpperFrequency';
					xAsIOAccWrite1.value := LIMIT(1,REAL_TO_UDINT(4.0*(MM2VIS.rF_VibSens_CenterBand2 + Para.rIdx_VibSens_BandWidth/2)),40000);
					ucWriteBandCnt		 := 0;

					(* Band 3 - Sensor 1 *)
				17: bWrite		 		 := TRUE;
					szWriteConfig		 := 'FrequencyBand03LowerFrequency';
					xAsIOAccWrite1.value := LIMIT(1,REAL_TO_UDINT(4.0*(MM2VIS.rF_VibSens_CenterBand3 - Para.rIdx_VibSens_BandWidth/2)),40000);
					ucWriteBandCnt		 := 18;
				18: bWrite		 		 := TRUE;
					szWriteConfig		 := 'FrequencyBand03UpperFrequency';
					xAsIOAccWrite1.value := LIMIT(1,REAL_TO_UDINT(4.0*(MM2VIS.rF_VibSens_CenterBand3 + Para.rIdx_VibSens_BandWidth/2)),40000);
					ucWriteBandCnt		 := 19;
					(* Band 3 - Sensor 2 *)
				19: bWrite		 		 := TRUE;
					szWriteConfig		 := 'FrequencyBand11LowerFrequency';
					xAsIOAccWrite1.value := LIMIT(1,REAL_TO_UDINT(4.0*(MM2VIS.rF_VibSens_CenterBand3 - Para.rIdx_VibSens_BandWidth/2)),40000);
					ucWriteBandCnt		 := 20;
				20: bWrite		 		 := TRUE;
					szWriteConfig		 := 'FrequencyBand11UpperFrequency';
					xAsIOAccWrite1.value := LIMIT(1,REAL_TO_UDINT(4.0*(MM2VIS.rF_VibSens_CenterBand3 + Para.rIdx_VibSens_BandWidth/2)),40000);
					ucWriteBandCnt		 := 21;
					(* Band 3 - Sensor 3 *)
				21: bWrite		 		 := TRUE;
					szWriteConfig		 := 'FrequencyBand19LowerFrequency';
					xAsIOAccWrite1.value := LIMIT(1,REAL_TO_UDINT(4.0*(MM2VIS.rF_VibSens_CenterBand3 - Para.rIdx_VibSens_BandWidth/2)),40000);
					ucWriteBandCnt		 := 22;
				22: bWrite		 		 := TRUE;
					szWriteConfig		 := 'FrequencyBand19UpperFrequency';
					xAsIOAccWrite1.value := LIMIT(1,REAL_TO_UDINT(4.0*(MM2VIS.rF_VibSens_CenterBand3 + Para.rIdx_VibSens_BandWidth/2)),40000);
					ucWriteBandCnt		 := 23;
					(* Band 3 - Sensor 4 *)
				23: bWrite		 		 := TRUE;
					szWriteConfig		 := 'FrequencyBand27LowerFrequency';
					xAsIOAccWrite1.value := LIMIT(1,REAL_TO_UDINT(4.0*(MM2VIS.rF_VibSens_CenterBand3 - Para.rIdx_VibSens_BandWidth/2)),40000);
					ucWriteBandCnt		 := 24;
				24: bWrite		 		 := TRUE;
					szWriteConfig		 := 'FrequencyBand27UpperFrequency';
					xAsIOAccWrite1.value := LIMIT(1,REAL_TO_UDINT(4.0*(MM2VIS.rF_VibSens_CenterBand3 + Para.rIdx_VibSens_BandWidth/2)),40000);
					ucWriteBandCnt		 := 0;

					(* Band 4 - Sensor 1 *)
				25: bWrite		 		 := TRUE;
					szWriteConfig		 := 'FrequencyBand04LowerFrequency';
					xAsIOAccWrite1.value := LIMIT(1,REAL_TO_UDINT(4.0*(MM2VIS.rF_VibSens_CenterBand4 - Para.rIdx_VibSens_BandWidth/2)),40000);
					ucWriteBandCnt		 := 26;
				26: bWrite		 		 := TRUE;
					szWriteConfig		 := 'FrequencyBand04UpperFrequency';
					xAsIOAccWrite1.value := LIMIT(1,REAL_TO_UDINT(4.0*(MM2VIS.rF_VibSens_CenterBand4 + Para.rIdx_VibSens_BandWidth/2)),40000);
					ucWriteBandCnt		 := 27;
					(* Band 4 - Sensor 2 *)
				27: bWrite		 		 := TRUE;
					szWriteConfig		 := 'FrequencyBand12LowerFrequency';
					xAsIOAccWrite1.value := LIMIT(1,REAL_TO_UDINT(4.0*(MM2VIS.rF_VibSens_CenterBand4 - Para.rIdx_VibSens_BandWidth/2)),40000);
					ucWriteBandCnt		 := 28;
				28: bWrite		 		 := TRUE;
					szWriteConfig		 := 'FrequencyBand12UpperFrequency';
					xAsIOAccWrite1.value := LIMIT(1,REAL_TO_UDINT(4.0*(MM2VIS.rF_VibSens_CenterBand4 + Para.rIdx_VibSens_BandWidth/2)),40000);
					ucWriteBandCnt		 := 29;
					(* Band 4 - Sensor 3 *)
				29: bWrite		 		 := TRUE;
					szWriteConfig		 := 'FrequencyBand20LowerFrequency';
					xAsIOAccWrite1.value := LIMIT(1,REAL_TO_UDINT(4.0*(MM2VIS.rF_VibSens_CenterBand4 - Para.rIdx_VibSens_BandWidth/2)),40000);
					ucWriteBandCnt		 := 30;
				30: bWrite		 		 := TRUE;
					szWriteConfig		 := 'FrequencyBand20UpperFrequency';
					xAsIOAccWrite1.value := LIMIT(1,REAL_TO_UDINT(4.0*(MM2VIS.rF_VibSens_CenterBand4 + Para.rIdx_VibSens_BandWidth/2)),40000);
					ucWriteBandCnt		 := 31;
					(* Band 4 - Sensor 4 *)
				31: bWrite		 		 := TRUE;
					szWriteConfig		 := 'FrequencyBand28LowerFrequency';
					xAsIOAccWrite1.value := LIMIT(1,REAL_TO_UDINT(4.0*(MM2VIS.rF_VibSens_CenterBand4 - Para.rIdx_VibSens_BandWidth/2)),40000);
					ucWriteBandCnt		 := 32;
				32: bWrite		 		 := TRUE;
					szWriteConfig		 := 'FrequencyBand28UpperFrequency';
					xAsIOAccWrite1.value := LIMIT(1,REAL_TO_UDINT(4.0*(MM2VIS.rF_VibSens_CenterBand4 + Para.rIdx_VibSens_BandWidth/2)),40000);
					ucWriteBandCnt		 := 0;

					(* Band 5 - Sensor 1 *)
				33: bWrite		 		 := TRUE;
					szWriteConfig		 := 'FrequencyBand05LowerFrequency';
					xAsIOAccWrite1.value := LIMIT(1,REAL_TO_UDINT(4.0*(MM2VIS.rF_VibSens_CenterBand5 - Para.rIdx_VibSens_BandWidth/2)),40000);
					ucWriteBandCnt		 := 34;
				34: bWrite		 		 := TRUE;
					szWriteConfig		 := 'FrequencyBand05UpperFrequency';
					xAsIOAccWrite1.value := LIMIT(1,REAL_TO_UDINT(4.0*(MM2VIS.rF_VibSens_CenterBand5 + Para.rIdx_VibSens_BandWidth/2)),40000);
					ucWriteBandCnt		 := 35;
					(* Band 5 - Sensor 2 *)
				35: bWrite		 		 := TRUE;
					szWriteConfig		 := 'FrequencyBand13LowerFrequency';
					xAsIOAccWrite1.value := LIMIT(1,REAL_TO_UDINT(4.0*(MM2VIS.rF_VibSens_CenterBand5 - Para.rIdx_VibSens_BandWidth/2)),40000);
					ucWriteBandCnt		 := 36;
				36: bWrite		 		 := TRUE;
					szWriteConfig		 := 'FrequencyBand13UpperFrequency';
					xAsIOAccWrite1.value := LIMIT(1,REAL_TO_UDINT(4.0*(MM2VIS.rF_VibSens_CenterBand5 + Para.rIdx_VibSens_BandWidth/2)),40000);
					ucWriteBandCnt		 := 37;
					(* Band 5 - Sensor 3 *)
				37: bWrite		 		 := TRUE;
					szWriteConfig		 := 'FrequencyBand21LowerFrequency';
					xAsIOAccWrite1.value := LIMIT(1,REAL_TO_UDINT(4.0*(MM2VIS.rF_VibSens_CenterBand5 - Para.rIdx_VibSens_BandWidth/2)),40000);
					ucWriteBandCnt		 := 38;
				38: bWrite		 		 := TRUE;
					szWriteConfig		 := 'FrequencyBand21UpperFrequency';
					xAsIOAccWrite1.value := LIMIT(1,REAL_TO_UDINT(4.0*(MM2VIS.rF_VibSens_CenterBand5 + Para.rIdx_VibSens_BandWidth/2)),40000);
					ucWriteBandCnt		 := 39;
					(* Band 5 - Sensor 4 *)
				39: bWrite		 		 := TRUE;
					szWriteConfig		 := 'FrequencyBand29LowerFrequency';
					xAsIOAccWrite1.value := LIMIT(1,REAL_TO_UDINT(4.0*(MM2VIS.rF_VibSens_CenterBand5 - Para.rIdx_VibSens_BandWidth/2)),40000);
					ucWriteBandCnt		 := 40;
				40: bWrite		 		 := TRUE;
					szWriteConfig		 := 'FrequencyBand29UpperFrequency';
					xAsIOAccWrite1.value := LIMIT(1,REAL_TO_UDINT(4.0*(MM2VIS.rF_VibSens_CenterBand5 + Para.rIdx_VibSens_BandWidth/2)),40000);
					ucWriteBandCnt		 := 0;

					(* Band 6 - Sensor 1 *)
				41: bWrite		 		 := TRUE;
					szWriteConfig		 := 'FrequencyBand06LowerFrequency';
					xAsIOAccWrite1.value := LIMIT(1,REAL_TO_UDINT(4.0*(MM2VIS.rF_VibSens_CenterBand6 - Para.rIdx_VibSens_BandWidth/2)),40000);
					ucWriteBandCnt		 := 42;
				42: bWrite		 		 := TRUE;
					szWriteConfig		 := 'FrequencyBand06UpperFrequency';
					xAsIOAccWrite1.value := LIMIT(1,REAL_TO_UDINT(4.0*(MM2VIS.rF_VibSens_CenterBand6 + Para.rIdx_VibSens_BandWidth/2)),40000);
					ucWriteBandCnt		 := 43;
					(* Band 6 - Sensor 2 *)
				43: bWrite		 		 := TRUE;
					szWriteConfig		 := 'FrequencyBand14LowerFrequency';
					xAsIOAccWrite1.value := LIMIT(1,REAL_TO_UDINT(4.0*(MM2VIS.rF_VibSens_CenterBand6 - Para.rIdx_VibSens_BandWidth/2)),40000);
					ucWriteBandCnt		 := 44;
				44: bWrite		 		 := TRUE;
					szWriteConfig		 := 'FrequencyBand14UpperFrequency';
					xAsIOAccWrite1.value := LIMIT(1,REAL_TO_UDINT(4.0*(MM2VIS.rF_VibSens_CenterBand6 + Para.rIdx_VibSens_BandWidth/2)),40000);
					ucWriteBandCnt		 := 45;
					(* Band 6 - Sensor 3 *)
				45: bWrite		 		 := TRUE;
					szWriteConfig		 := 'FrequencyBand22LowerFrequency';
					xAsIOAccWrite1.value := LIMIT(1,REAL_TO_UDINT(4.0*(MM2VIS.rF_VibSens_CenterBand6 - Para.rIdx_VibSens_BandWidth/2)),40000);
					ucWriteBandCnt		 := 46;
				46: bWrite		 		 := TRUE;
					szWriteConfig		 := 'FrequencyBand22UpperFrequency';
					xAsIOAccWrite1.value := LIMIT(1,REAL_TO_UDINT(4.0*(MM2VIS.rF_VibSens_CenterBand6 + Para.rIdx_VibSens_BandWidth/2)),40000);
					ucWriteBandCnt		 := 47;
					(* Band 6 - Sensor 4 *)
				47: bWrite		 		 := TRUE;
					szWriteConfig		 := 'FrequencyBand30LowerFrequency';
					xAsIOAccWrite1.value := LIMIT(1,REAL_TO_UDINT(4.0*(MM2VIS.rF_VibSens_CenterBand6 - Para.rIdx_VibSens_BandWidth/2)),40000);
					ucWriteBandCnt		 := 48;
				48: bWrite		 		 := TRUE;
					szWriteConfig		 := 'FrequencyBand30UpperFrequency';
					xAsIOAccWrite1.value := LIMIT(1,REAL_TO_UDINT(4.0*(MM2VIS.rF_VibSens_CenterBand6 + Para.rIdx_VibSens_BandWidth/2)),40000);
					ucWriteBandCnt		 := 0;

					(* Band 7 - Sensor 1 *)
				49: bWrite		 		 := TRUE;
					szWriteConfig		 := 'FrequencyBand07LowerFrequency';
					xAsIOAccWrite1.value := LIMIT(1,REAL_TO_UDINT(4.0*(MM2VIS.rF_VibSens_CenterBand7 - Para.rIdx_VibSens_BandWidth/2)),40000);
					ucWriteBandCnt		 := 50;
				50: bWrite		 		 := TRUE;
					szWriteConfig		 := 'FrequencyBand07UpperFrequency';
					xAsIOAccWrite1.value := LIMIT(1,REAL_TO_UDINT(4.0*(MM2VIS.rF_VibSens_CenterBand7 + Para.rIdx_VibSens_BandWidth/2)),40000);
					ucWriteBandCnt		 := 51;
					(* Band 7 - Sensor 2 *)
				51: bWrite		 		 := TRUE;
					szWriteConfig		 := 'FrequencyBand15LowerFrequency';
					xAsIOAccWrite1.value := LIMIT(1,REAL_TO_UDINT(4.0*(MM2VIS.rF_VibSens_CenterBand7 - Para.rIdx_VibSens_BandWidth/2)),40000);
					ucWriteBandCnt		 := 52;
				52: bWrite		 		 := TRUE;
					szWriteConfig		 := 'FrequencyBand15UpperFrequency';
					xAsIOAccWrite1.value := LIMIT(1,REAL_TO_UDINT(4.0*(MM2VIS.rF_VibSens_CenterBand7 + Para.rIdx_VibSens_BandWidth/2)),40000);
					ucWriteBandCnt		 := 53;
					(* Band 7 - Sensor 3 *)
				53: bWrite		 		 := TRUE;
					szWriteConfig		 := 'FrequencyBand23LowerFrequency';
					xAsIOAccWrite1.value := LIMIT(1,REAL_TO_UDINT(4.0*(MM2VIS.rF_VibSens_CenterBand7 - Para.rIdx_VibSens_BandWidth/2)),40000);
					ucWriteBandCnt		 := 54;
				54: bWrite		 		 := TRUE;
					szWriteConfig		 := 'FrequencyBand23UpperFrequency';
					xAsIOAccWrite1.value := LIMIT(1,REAL_TO_UDINT(4.0*(MM2VIS.rF_VibSens_CenterBand7 + Para.rIdx_VibSens_BandWidth/2)),40000);
					ucWriteBandCnt		 := 55;
					(* Band 7 - Sensor 4 *)
				55: bWrite		 		 := TRUE;
					szWriteConfig		 := 'FrequencyBand31LowerFrequency';
					xAsIOAccWrite1.value := LIMIT(1,REAL_TO_UDINT(4.0*(MM2VIS.rF_VibSens_CenterBand7 - Para.rIdx_VibSens_BandWidth/2)),40000);
					ucWriteBandCnt		 := 56;
				56: bWrite		 		 := TRUE;
					szWriteConfig		 := 'FrequencyBand31UpperFrequency';
					xAsIOAccWrite1.value := LIMIT(1,REAL_TO_UDINT(4.0*(MM2VIS.rF_VibSens_CenterBand7 + Para.rIdx_VibSens_BandWidth/2)),40000);
					ucWriteBandCnt		 := 0;

					(* Band 8 - Sensor 1 *)
				57: bWrite		 		 := TRUE;
					szWriteConfig		 := 'FrequencyBand08LowerFrequency';
					xAsIOAccWrite1.value := LIMIT(1,REAL_TO_UDINT(4.0*(MM2VIS.rF_VibSens_CenterBand8 - Para.rIdx_VibSens_BandWidth/2)),40000);
					ucWriteBandCnt		 := 58;
				58: bWrite		 		 := TRUE;
					szWriteConfig		 := 'FrequencyBand08UpperFrequency';
					xAsIOAccWrite1.value := LIMIT(1,REAL_TO_UDINT(4.0*(MM2VIS.rF_VibSens_CenterBand8 + Para.rIdx_VibSens_BandWidth/2)),40000);
					ucWriteBandCnt		 := 59;
					(* Band 8 - Sensor 2 *)
				59: bWrite		 		 := TRUE;
					szWriteConfig		 := 'FrequencyBand16LowerFrequency';
					xAsIOAccWrite1.value := LIMIT(1,REAL_TO_UDINT(4.0*(MM2VIS.rF_VibSens_CenterBand8 - Para.rIdx_VibSens_BandWidth/2)),40000);
					ucWriteBandCnt		 := 60;
				60: bWrite		 		 := TRUE;
					szWriteConfig		 := 'FrequencyBand16UpperFrequency';
					xAsIOAccWrite1.value := LIMIT(1,REAL_TO_UDINT(4.0*(MM2VIS.rF_VibSens_CenterBand8 + Para.rIdx_VibSens_BandWidth/2)),40000);
					ucWriteBandCnt		 := 61;
					(* Band 8 - Sensor 3 *)
				61: bWrite		 		 := TRUE;
					szWriteConfig		 := 'FrequencyBand24LowerFrequency';
					xAsIOAccWrite1.value := LIMIT(1,REAL_TO_UDINT(4.0*(MM2VIS.rF_VibSens_CenterBand8 - Para.rIdx_VibSens_BandWidth/2)),40000);
					ucWriteBandCnt		 := 62;
				62: bWrite		 		 := TRUE;
					szWriteConfig		 := 'FrequencyBand24UpperFrequency';
					xAsIOAccWrite1.value := LIMIT(1,REAL_TO_UDINT(4.0*(MM2VIS.rF_VibSens_CenterBand8 + Para.rIdx_VibSens_BandWidth/2)),40000);
					ucWriteBandCnt		 := 63;
					(* Band 8 - Sensor 4 *)
				63: bWrite		 		 := TRUE;
					szWriteConfig		 := 'FrequencyBand32LowerFrequency';
					xAsIOAccWrite1.value := LIMIT(1,REAL_TO_UDINT(4.0*(MM2VIS.rF_VibSens_CenterBand8 - Para.rIdx_VibSens_BandWidth/2)),40000);
					ucWriteBandCnt		 := 64;
				64: bWrite		 		 := TRUE;
					szWriteConfig		 := 'FrequencyBand32UpperFrequency';
					xAsIOAccWrite1.value := LIMIT(1,REAL_TO_UDINT(4.0*(MM2VIS.rF_VibSens_CenterBand8 + Para.rIdx_VibSens_BandWidth/2)),40000);
					ucWriteBandCnt		 := 0;

			END_CASE;

		END_IF;

		(* read & write X204810 registers *)

		(* write band configuration and miscellaneous values *)
		IF bWrite THEN														(* set bWrite to TRUE to write a register on the CM48810 X20 module *)
			xAsIOAccWrite1.enable	    := TRUE;
			xAsIOAccWrite1.pDeviceName  := xCM4810.paramMain.pModulePath;
//			xAsIOAccWrite1.value	    := 0;								(* set value to write at this attribute of the function block *)
			xAsIOAccWrite1.pChannelName	:= ADR(szWriteConfig);				(* set name of register to write at string pv szWriteConfig *)
			xAsIOAccWrite1();

			IF xAsIOAccWrite1.status = 0 THEN
				bWrite := FALSE;
			END_IF;
		END_IF;

		(* read miscellaneous values *)
		IF bRead THEN														(* set bRead to TRUE to read a register from the CM48810 X20 module *)
			xAsIOAccRead1.enable	   := TRUE;
			xAsIOAccRead1.pDeviceName  := xCM4810.paramMain.pModulePath;
//			xAsIOAccRead1.value;											(* here the read valure can be found *)
			xAsIOAccRead1.pChannelName := ADR(szReadConfig);				(* set name of register to read at string pv szReadConfig *)
			xAsIOAccRead1();

			IF xAsIOAccRead1.status = 0 THEN
				bRead := FALSE;
			END_IF;
		END_IF;

	END_IF;

END_PROGRAM
```
